LIN {X 0,Y 523.443,Z 553.477,A -85,B 0,C 180,E1 -4766.15,E2 -4766.15} C_VEL
LIN {X 0,Y 523.367,Z 555.34,A -85,B 0,C 180,E1 -4766.921,E2 -4766.921} C_VEL
LIN {X 0,Y 523.334,Z 556.738,A -85,B 0,C 180,E1 -4767.691,E2 -4767.691} C_VEL
LIN {X 0,Y 523.25,Z 558.344,A -85,B 0,C 180,E1 -4769.23,E2 -4769.23} C_VEL
LIN {X 0,Y 523.25,Z 558.561,A -85,B 0,C 180,E1 -4770,E2 -4770} C_VEL
LIN {X 0,Y 523.274,Z 557.739,A -85,B 0,C 180,E1 -4771.539,E2 -4771.539} C_VEL
LIN {X 0,Y 523.334,Z 556.745,A -85,B 0,C 180,E1 -4772.309,E2 -4772.309} C_VEL
LIN {X 0,Y 523.367,Z 555.349,A -85,B 0,C 180,E1 -4773.079,E2 -4773.079} C_VEL
LIN {X 0,Y 523.424,Z 552.411,A -85,B 0,C 180,E1 -4774.235,E2 -4774.235} C_VEL
LIN {X 0,Y 523.461,Z 548.432,A -85,B 0,C 180,E1 -4775.392,E2 -4775.392} C_VEL
LIN {X 0,Y 523.514,Z 543.213,A -85,B 0,C 180,E1 -4776.572,E2 -4776.572} C_VEL
LIN {X 0,Y 523.646,Z 536.865,A -85,B 0,C 180,E1 -4777.713,E2 -4777.713} C_VEL
LIN {X 0,Y 523.815,Z 528.823,A -85,B 0,C 180,E1 -4778.876,E2 -4778.876} C_VEL
LIN {X 0,Y 524.043,Z 520.63,A -85,B 0,C 180,E1 -4779.845,E2 -4779.845} C_VEL
LIN {X 0,Y 524.325,Z 510.642,A -85,B 0,C 180,E1 -4780.816,E2 -4780.816} C_VEL
LIN {X 0,Y 524.62,Z 499.343,A -85,B 0,C 180,E1 -4781.691,E2 -4781.691} C_VEL
LIN {X 0,Y 524.85,Z 488.315,A -85,B 0,C 180,E1 -4782.371,E2 -4782.371} C_VEL
LIN {X 0,Y 525.116,Z 476.074,A -85,B 0,C 180,E1 -4782.954,E2 -4782.954} C_VEL
LIN {X 0,Y 525.355,Z 463.228,A -85,B 0,C 180,E1 -4783.391,E2 -4783.391} C_VEL
LIN {X 0,Y 525.545,Z 449.606,A -85,B 0,C 180,E1 -4783.681,E2 -4783.681} C_VEL
LIN {X 0,Y 525.885,Z 356.541,A -85,B 0,C 180,E1 -4784.961,E2 -4784.961} C_VEL
LIN {X 0,Y 524.307,Z 345.556,A -85,B 0,C 180,E1 -4785.178,E2 -4785.178} C_VEL
LIN {X 0,Y 524.738,Z 323.578,A -85,B 0,C 180,E1 -4788.527,E2 -4788.527} C_VEL
LIN {X 0,Y 525.158,Z 305.074,A -85,B 0,C 180,E1 -4791.387,E2 -4791.387} C_VEL
LIN {X 0,Y 525.431,Z 293.248,A -85,B 0,C 180,E1 -4793.239,E2 -4793.239} C_VEL
LIN {X 0,Y 524.002,Z 285.214,A -85,B 0,C 180,E1 -4794.594,E2 -4794.594} C_VEL
LIN {X 0,Y 523.979,Z 285.218,A -85,B 0,C 180,E1 -4797.718,E2 -4797.718} C_VEL
LIN {X 0,Y 523.945,Z 285.215,A -85,B 0,C 180,E1 -4800.854,E2 -4800.854} C_VEL
LIN {X 0,Y 523.959,Z 285.215,A -85,B 0,C 180,E1 -4803.734,E2 -4803.734} C_VEL
LIN {X 0,Y 523.903,Z 285.227,A -85,B 0,C 180,E1 -4806.401,E2 -4806.401} C_VEL
LIN {X 0,Y 523.919,Z 285.218,A -85,B 0,C 180,E1 -4809.084,E2 -4809.084} C_VEL
LIN {X 0,Y 523.953,Z 285.218,A -85,B 0,C 180,E1 -4812.118,E2 -4812.118} C_VEL
LIN {X 0,Y 523.942,Z 285.215,A -85,B 0,C 180,E1 -4815.309,E2 -4815.309} C_VEL
LIN {X 0,Y 523.957,Z 285.221,A -85,B 0,C 180,E1 -4818.689,E2 -4818.689} C_VEL
LIN {X 0,Y 523.914,Z 285.221,A -85,B 0,C 180,E1 -4821.08,E2 -4821.08} C_VEL
LIN {X 0,Y 523.898,Z 285.22,A -85,B 0,C 180,E1 -4823.825,E2 -4823.825} C_VEL
LIN {X 0,Y 523.938,Z 285.222,A -85,B 0,C 180,E1 -4826.635,E2 -4826.635} C_VEL
LIN {X 0,Y 523.953,Z 285.216,A -85,B 0,C 180,E1 -4829.355,E2 -4829.355} C_VEL
LIN {X 0,Y 523.975,Z 285.211,A -85,B 0,C 180,E1 -4832.281,E2 -4832.281} C_VEL
LIN {X 0,Y 523.949,Z 285.217,A -85,B 0,C 180,E1 -4834.581,E2 -4834.581} C_VEL
LIN {X 0,Y 523.913,Z 285.228,A -85,B 0,C 180,E1 -4837.106,E2 -4837.106} C_VEL
LIN {X 0,Y 523.974,Z 285.211,A -85,B 0,C 180,E1 -4839.866,E2 -4839.866} C_VEL
LIN {X 0,Y 523.962,Z 285.215,A -85,B 0,C 180,E1 -4842.837,E2 -4842.837} C_VEL
LIN {X 0,Y 524,Z 285.216,A -85,B 0,C 180,E1 -4845.236,E2 -4845.236} C_VEL
LIN {X 0,Y 524.007,Z 285.206,A -85,B 0,C 180,E1 -4848.394,E2 -4848.394} C_VEL
LIN {X 0,Y 524,Z 285.217,A -85,B 0,C 180,E1 -4851.516,E2 -4851.516} C_VEL
LIN {X 0,Y 524.076,Z 285.198,A -85,B 0,C 180,E1 -4854.613,E2 -4854.613} C_VEL
LIN {X 0,Y 524.104,Z 285.204,A -85,B 0,C 180,E1 -4857.694,E2 -4857.694} C_VEL
LIN {X 0,Y 524.116,Z 285.193,A -85,B 0,C 180,E1 -4860.768,E2 -4860.768} C_VEL
LIN {X 0,Y 524.067,Z 285.2,A -85,B 0,C 180,E1 -4863.075,E2 -4863.075} C_VEL
LIN {X 0,Y 524.023,Z 285.21,A -85,B 0,C 180,E1 -4866.159,E2 -4866.159} C_VEL
LIN {X 0,Y 523.998,Z 285.21,A -85,B 0,C 180,E1 -4868.484,E2 -4868.484} C_VEL
LIN {X 0,Y 523.997,Z 285.213,A -85,B 0,C 180,E1 -4871.739,E2 -4871.739} C_VEL
LIN {X 0,Y 523.986,Z 285.209,A -85,B 0,C 180,E1 -4875.052,E2 -4875.052} C_VEL
LIN {X 0,Y 523.941,Z 285.22,A -85,B 0,C 180,E1 -4877.97,E2 -4877.97} C_VEL
LIN {X 0,Y 523.966,Z 285.219,A -85,B 0,C 180,E1 -4880.41,E2 -4880.41} C_VEL
LIN {X 0,Y 523.904,Z 285.221,A -85,B 0,C 180,E1 -4882.894,E2 -4882.894} C_VEL
LIN {X 0,Y 523.977,Z 285.214,A -85,B 0,C 180,E1 -4886.02,E2 -4886.02} C_VEL
LIN {X 0,Y 523.927,Z 285.22,A -85,B 0,C 180,E1 -4888.875,E2 -4888.875} C_VEL
LIN {X 0,Y 523.915,Z 285.218,A -85,B 0,C 180,E1 -4891.544,E2 -4891.544} C_VEL
LIN {X 0,Y 523.927,Z 285.22,A -85,B 0,C 180,E1 -4894.291,E2 -4894.291} C_VEL
LIN {X 0,Y 523.901,Z 285.223,A -85,B 0,C 180,E1 -4897.133,E2 -4897.133} C_VEL
LIN {X 0,Y 523.933,Z 285.216,A -85,B 0,C 180,E1 -4900.13,E2 -4900.13} C_VEL
LIN {X 0,Y 523.93,Z 285.219,A -85,B 0,C 180,E1 -4902.459,E2 -4902.459} C_VEL
LIN {X 0,Y 523.948,Z 285.218,A -85,B 0,C 180,E1 -4905.31,E2 -4905.31} C_VEL
LIN {X 0,Y 523.891,Z 285.227,A -85,B 0,C 180,E1 -4906.893,E2 -4906.893} C_VEL
LIN {X 0,Y 523.211,Z 285.309,A -85,B 0,C 180,E1 -4907.535,E2 -4907.535} C_VEL
LIN {X 0,Y 520.359,Z 285.664,A -85,B 0,C 180,E1 -4908.576,E2 -4908.576} C_VEL
LIN {X 0,Y 517.961,Z 285.964,A -85,B 0,C 180,E1 -4909.415,E2 -4909.415} C_VEL
LIN {X 0,Y 516.935,Z 286.088,A -85,B 0,C 180,E1 -4910.063,E2 -4910.063} C_VEL
LIN {X 0,Y 516.854,Z 286.098,A -85,B 0,C 180,E1 -4910.282,E2 -4910.282} C_VEL
LIN {X 0,Y 516.873,Z 286.102,A -85,B 0,C 180,E1 -4913.344,E2 -4913.344} C_VEL
LIN {X 0,Y 516.88,Z 286.094,A -85,B 0,C 180,E1 -4916.119,E2 -4916.119} C_VEL
LIN {X 0,Y 516.885,Z 286.097,A -85,B 0,C 180,E1 -4918.937,E2 -4918.937} C_VEL
LIN {X 0,Y 516.855,Z 286.104,A -85,B 0,C 180,E1 -4921.582,E2 -4921.582} C_VEL
LIN {X 0,Y 516.865,Z 286.097,A -85,B 0,C 180,E1 -4924.208,E2 -4924.208} C_VEL
LIN {X 0,Y 516.855,Z 286.098,A -85,B 0,C 180,E1 -4926.776,E2 -4926.776} C_VEL
LIN {X 0,Y 516.938,Z 286.095,A -85,B 0,C 180,E1 -4929.732,E2 -4929.732} C_VEL
LIN {X 0,Y 516.883,Z 286.094,A -85,B 0,C 180,E1 -4932.595,E2 -4932.595} C_VEL
LIN {X 0,Y 516.941,Z 286.087,A -85,B 0,C 180,E1 -4935.031,E2 -4935.031} C_VEL
LIN {X 0,Y 516.925,Z 286.096,A -85,B 0,C 180,E1 -4938.233,E2 -4938.233} C_VEL
LIN {X 0,Y 516.906,Z 286.192,A -85,B 0,C 180,E1 -4940.289,E2 -4940.289} C_VEL
LIN {X 0,Y 517.467,Z 290.917,A -85,B 0,C 180,E1 -4941.212,E2 -4941.212} C_VEL
LIN {X 0,Y 517.225,Z 306.513,A -85,B 0,C 180,E1 -4944.151,E2 -4944.151} C_VEL
LIN {X 0,Y 517.209,Z 309.369,A -85,B 0,C 180,E1 -4944.689,E2 -4944.689} C_VEL
LIN {X 0,Y 519.108,Z 320.246,A -85,B 0,C 180,E1 -4944.903,E2 -4944.903} C_VEL
LIN {X 0,Y 518.613,Z 416.523,A -85,B 0,C 180,E1 -4946.261,E2 -4946.261} C_VEL
LIN {X 0,Y 518.43,Z 429.494,A -85,B 0,C 180,E1 -4946.6,E2 -4946.6} C_VEL
LIN {X 0,Y 518.257,Z 441.97,A -85,B 0,C 180,E1 -4947.085,E2 -4947.085} C_VEL
LIN {X 0,Y 517.976,Z 453.153,A -85,B 0,C 180,E1 -4947.667,E2 -4947.667} C_VEL
LIN {X 0,Y 517.599,Z 464.695,A -85,B 0,C 180,E1 -4948.444,E2 -4948.444} C_VEL
LIN {X 0,Y 517.235,Z 475.076,A -85,B 0,C 180,E1 -4949.319,E2 -4949.319} C_VEL
LIN {X 0,Y 517.081,Z 483.55,A -85,B 0,C 180,E1 -4950.195,E2 -4950.195} C_VEL
LIN {X 0,Y 516.841,Z 491.401,A -85,B 0,C 180,E1 -4951.169,E2 -4951.169} C_VEL
LIN {X 0,Y 516.597,Z 499.125,A -85,B 0,C 180,E1 -4952.339,E2 -4952.339} C_VEL
LIN {X 0,Y 516.472,Z 505.306,A -85,B 0,C 180,E1 -4953.511,E2 -4953.511} C_VEL
LIN {X 0,Y 516.328,Z 510.245,A -85,B 0,C 180,E1 -4954.685,E2 -4954.685} C_VEL
LIN {X 0,Y 516.374,Z 514.064,A -85,B 0,C 180,E1 -4955.859,E2 -4955.859} C_VEL
LIN {X 0,Y 516.281,Z 516.886,A -85,B 0,C 180,E1 -4957.037,E2 -4957.037} C_VEL
LIN {X 0,Y 516.266,Z 518.217,A -85,B 0,C 180,E1 -4957.824,E2 -4957.824} C_VEL
LIN {X 0,Y 516.212,Z 519.159,A -85,B 0,C 180,E1 -4958.613,E2 -4958.613} C_VEL
LIN {X 0,Y 516.175,Z 519.709,A -85,B 0,C 180,E1 -4959.404,E2 -4959.404} C_VEL
LIN {X 0,Y 516.236,Z 519.817,A -85,B 0,C 180,E1 -4960.194,E2 -4960.194} C_VEL
LIN {X 0,Y 516.281,Z 519.192,A -85,B 0,C 180,E1 -4961.445,E2 -4961.445} C_VEL
LIN {X 0,Y 516.223,Z 517.759,A -85,B 0,C 180,E1 -4962.582,E2 -4962.582} C_VEL
LIN {X 0,Y 516.234,Z 516.198,A -85,B 0,C 180,E1 -4963.382,E2 -4963.382} C_VEL
LIN {X 0,Y 516.359,Z 513.134,A -85,B 0,C 180,E1 -4964.553,E2 -4964.553} C_VEL
LIN {X 0,Y 516.416,Z 508.746,A -85,B 0,C 180,E1 -4965.794,E2 -4965.794} C_VEL
LIN {X 0,Y 516.554,Z 503.194,A -85,B 0,C 180,E1 -4967.009,E2 -4967.009} C_VEL
LIN {X 0,Y 516.753,Z 496.184,A -85,B 0,C 180,E1 -4968.229,E2 -4968.229} C_VEL
LIN {X 0,Y 516.9,Z 488.946,A -85,B 0,C 180,E1 -4969.252,E2 -4969.252} C_VEL
LIN {X 0,Y 517.195,Z 479.415,A -85,B 0,C 180,E1 -4970.345,E2 -4970.345} C_VEL
LIN {X 0,Y 517.499,Z 469.068,A -85,B 0,C 180,E1 -4971.302,E2 -4971.302} C_VEL
LIN {X 0,Y 517.853,Z 457.976,A -85,B 0,C 180,E1 -4972.124,E2 -4972.124} C_VEL
LIN {X 0,Y 518.12,Z 446.531,A -85,B 0,C 180,E1 -4972.787,E2 -4972.787} C_VEL
LIN {X 0,Y 518.289,Z 434.594,A -85,B 0,C 180,E1 -4973.315,E2 -4973.315} C_VEL
LIN {X 0,Y 518.439,Z 421.216,A -85,B 0,C 180,E1 -4973.731,E2 -4973.731} C_VEL
LIN {X 0,Y 518.604,Z 406.66,A -85,B 0,C 180,E1 -4973.989,E2 -4973.989} C_VEL
LIN {X 0,Y 519.054,Z 319.507,A -85,B 0,C 180,E1 -4975.2,E2 -4975.2} C_VEL
LIN {X 0,Y 517.236,Z 309.202,A -85,B 0,C 180,E1 -4975.422,E2 -4975.422} C_VEL
LIN {X 0,Y 517.357,Z 293.041,A -85,B 0,C 180,E1 -4978.389,E2 -4978.389} C_VEL
LIN {X 0,Y 517.28,Z 288.195,A -85,B 0,C 180,E1 -4979.282,E2 -4979.282} C_VEL
LIN {X 0,Y 516.952,Z 286.097,A -85,B 0,C 180,E1 -4979.697,E2 -4979.697} C_VEL
LIN {X 0,Y 516.894,Z 286.096,A -85,B 0,C 180,E1 -4982.947,E2 -4982.947} C_VEL
LIN {X 0,Y 516.871,Z 286.099,A -85,B 0,C 180,E1 -4985.78,E2 -4985.78} C_VEL
LIN {X 0,Y 516.879,Z 286.102,A -85,B 0,C 180,E1 -4988.716,E2 -4988.716} C_VEL
LIN {X 0,Y 516.911,Z 286.092,A -85,B 0,C 180,E1 -4991.775,E2 -4991.775} C_VEL
LIN {X 0,Y 516.894,Z 286.098,A -85,B 0,C 180,E1 -4995.007,E2 -4995.007} C_VEL
LIN {X 0,Y 516.912,Z 286.095,A -85,B 0,C 180,E1 -4998.399,E2 -4998.399} C_VEL
LIN {X 0,Y 516.88,Z 286.097,A -85,B 0,C 180,E1 -5001.284,E2 -5001.284} C_VEL
LIN {X 0,Y 516.87,Z 286.095,A -85,B 0,C 180,E1 -5004.22,E2 -5004.22} C_VEL
LIN {X 0,Y 516.894,Z 286.1,A -85,B 0,C 180,E1 -5007.053,E2 -5007.053} C_VEL
LIN {X 0,Y 516.891,Z 286.092,A -85,B 0,C 180,E1 -5009.796,E2 -5009.796} C_VEL
LIN {X 0,Y 516.925,Z 286.087,A -85,B 0,C 180,E1 -5012.467,E2 -5012.467} C_VEL
LIN {X 0,Y 516.908,Z 286.096,A -85,B 0,C 180,E1 -5015.072,E2 -5015.072} C_VEL
LIN {X 0,Y 516.884,Z 286.093,A -85,B 0,C 180,E1 -5018.462,E2 -5018.462} C_VEL
LIN {X 0,Y 516.9,Z 286.092,A -85,B 0,C 180,E1 -5020.955,E2 -5020.955} C_VEL
LIN {X 0,Y 516.913,Z 286.099,A -85,B 0,C 180,E1 -5023.41,E2 -5023.41} C_VEL
LIN {X 0,Y 516.894,Z 286.099,A -85,B 0,C 180,E1 -5025.834,E2 -5025.834} C_VEL
LIN {X 0,Y 516.965,Z 286.084,A -85,B 0,C 180,E1 -5028.234,E2 -5028.234} C_VEL
LIN {X 0,Y 516.967,Z 286.088,A -85,B 0,C 180,E1 -5031.4,E2 -5031.4} C_VEL
LIN {X 0,Y 517.001,Z 286.086,A -85,B 0,C 180,E1 -5033.757,E2 -5033.757} C_VEL
LIN {X 0,Y 517.012,Z 286.077,A -85,B 0,C 180,E1 -5036.883,E2 -5036.883} C_VEL
LIN {X 0,Y 517.085,Z 286.077,A -85,B 0,C 180,E1 -5040,E2 -5040} C_VEL
LIN {X 0,Y 517.012,Z 286.076,A -85,B 0,C 180,E1 -5043.117,E2 -5043.117} C_VEL
LIN {X 0,Y 517.002,Z 286.085,A -85,B 0,C 180,E1 -5046.243,E2 -5046.243} C_VEL
LIN {X 0,Y 516.951,Z 286.085,A -85,B 0,C 180,E1 -5049.389,E2 -5049.389} C_VEL
LIN {X 0,Y 516.951,Z 286.084,A -85,B 0,C 180,E1 -5051.807,E2 -5051.807} C_VEL
LIN {X 0,Y 516.944,Z 286.086,A -85,B 0,C 180,E1 -5055.147,E2 -5055.147} C_VEL
LIN {X 0,Y 516.924,Z 286.092,A -85,B 0,C 180,E1 -5058.222,E2 -5058.222} C_VEL
LIN {X 0,Y 516.912,Z 286.097,A -85,B 0,C 180,E1 -5060.702,E2 -5060.702} C_VEL
LIN {X 0,Y 516.904,Z 286.092,A -85,B 0,C 180,E1 -5064.073,E2 -5064.073} C_VEL
LIN {X 0,Y 516.925,Z 286.095,A -85,B 0,C 180,E1 -5066.658,E2 -5066.658} C_VEL
LIN {X 0,Y 516.911,Z 286.092,A -85,B 0,C 180,E1 -5069.524,E2 -5069.524} C_VEL
LIN {X 0,Y 516.896,Z 286.094,A -85,B 0,C 180,E1 -5072.544,E2 -5072.544} C_VEL
LIN {X 0,Y 516.866,Z 286.101,A -85,B 0,C 180,E1 -5075.33,E2 -5075.33} C_VEL
LIN {X 0,Y 516.881,Z 286.095,A -85,B 0,C 180,E1 -5077.943,E2 -5077.943} C_VEL
LIN {X 0,Y 516.884,Z 286.09,A -85,B 0,C 180,E1 -5080.742,E2 -5080.742} C_VEL
LIN {X 0,Y 516.883,Z 286.096,A -85,B 0,C 180,E1 -5082.832,E2 -5082.832} C_VEL
LIN {X 0,Y 516.896,Z 286.095,A -85,B 0,C 180,E1 -5085.007,E2 -5085.007} C_VEL
LIN {X 0,Y 516.915,Z 286.091,A -85,B 0,C 180,E1 -5088.399,E2 -5088.399} C_VEL
LIN {X 0,Y 516.882,Z 286.099,A -85,B 0,C 180,E1 -5091.284,E2 -5091.284} C_VEL
LIN {X 0,Y 516.873,Z 286.099,A -85,B 0,C 180,E1 -5094.22,E2 -5094.22} C_VEL
LIN {X 0,Y 516.897,Z 286.095,A -85,B 0,C 180,E1 -5097.053,E2 -5097.053} C_VEL
LIN {X 0,Y 516.895,Z 286.101,A -85,B 0,C 180,E1 -5099.796,E2 -5099.796} C_VEL
LIN {X 0,Y 516.926,Z 286.093,A -85,B 0,C 180,E1 -5102.467,E2 -5102.467} C_VEL
LIN {X 0,Y 516.938,Z 286.123,A -85,B 0,C 180,E1 -5105.295,E2 -5105.295} C_VEL
LIN {X 0,Y 518.392,Z 294.033,A -85,B 0,C 180,E1 -5106.637,E2 -5106.637} C_VEL
LIN {X 0,Y 518.071,Z 309.859,A -85,B 0,C 180,E1 -5109.139,E2 -5109.139} C_VEL
LIN {X 0,Y 517.59,Z 329.884,A -85,B 0,C 180,E1 -5112.251,E2 -5112.251} C_VEL
LIN {X 0,Y 517.286,Z 345.547,A -85,B 0,C 180,E1 -5114.634,E2 -5114.634} C_VEL
LIN {X 0,Y 519.046,Z 357.722,A -85,B 0,C 180,E1 -5114.858,E2 -5114.858} C_VEL
LIN {X 0,Y 518.595,Z 453.618,A -85,B 0,C 180,E1 -5116.206,E2 -5116.206} C_VEL
LIN {X 0,Y 518.365,Z 466.951,A -85,B 0,C 180,E1 -5116.549,E2 -5116.549} C_VEL
LIN {X 0,Y 518.053,Z 480.278,A -85,B 0,C 180,E1 -5117.065,E2 -5117.065} C_VEL
LIN {X 0,Y 517.807,Z 492.339,A -85,B 0,C 180,E1 -5117.711,E2 -5117.711} C_VEL
LIN {X 0,Y 517.514,Z 504.391,A -85,B 0,C 180,E1 -5118.544,E2 -5118.544} C_VEL
LIN {X 0,Y 517.17,Z 514.61,A -85,B 0,C 180,E1 -5119.429,E2 -5119.429} C_VEL
LIN {X 0,Y 516.891,Z 523.806,A -85,B 0,C 180,E1 -5120.412,E2 -5120.412} C_VEL
LIN {X 0,Y 516.658,Z 532.769,A -85,B 0,C 180,E1 -5121.591,E2 -5121.591} C_VEL
LIN {X 0,Y 516.505,Z 539.985,A -85,B 0,C 180,E1 -5122.769,E2 -5122.769} C_VEL
LIN {X 0,Y 516.419,Z 546.558,A -85,B 0,C 180,E1 -5124.141,E2 -5124.141} C_VEL
LIN {X 0,Y 516.269,Z 550.903,A -85,B 0,C 180,E1 -5125.315,E2 -5125.315} C_VEL
LIN {X 0,Y 516.352,Z 553.21,A -85,B 0,C 180,E1 -5126.098,E2 -5126.098} C_VEL
LIN {X 0,Y 516.282,Z 555.074,A -85,B 0,C 180,E1 -5126.878,E2 -5126.878} C_VEL
LIN {X 0,Y 516.261,Z 556.473,A -85,B 0,C 180,E1 -5127.659,E2 -5127.659} C_VEL
LIN {X 0,Y 516.16,Z 558.079,A -85,B 0,C 180,E1 -5129.22,E2 -5129.22} C_VEL
LIN {X 0,Y 516.158,Z 558.297,A -85,B 0,C 180,E1 -5130,E2 -5130} C_VEL
LIN {X 0,Y 516.191,Z 557.476,A -85,B 0,C 180,E1 -5131.56,E2 -5131.56} C_VEL
LIN {X 0,Y 516.26,Z 556.482,A -85,B 0,C 180,E1 -5132.34,E2 -5132.34} C_VEL
LIN {X 0,Y 516.282,Z 555.086,A -85,B 0,C 180,E1 -5133.121,E2 -5133.121} C_VEL
LIN {X 0,Y 516.312,Z 552.147,A -85,B 0,C 180,E1 -5134.293,E2 -5134.293} C_VEL
LIN {X 0,Y 516.375,Z 548.168,A -85,B 0,C 180,E1 -5135.467,E2 -5135.467} C_VEL
LIN {X 0,Y 516.45,Z 542.253,A -85,B 0,C 180,E1 -5136.798,E2 -5136.798} C_VEL
LIN {X 0,Y 516.597,Z 535.359,A -85,B 0,C 180,E1 -5138.015,E2 -5138.015} C_VEL
LIN {X 0,Y 516.811,Z 527.063,A -85,B 0,C 180,E1 -5139.194,E2 -5139.194} C_VEL
LIN {X 0,Y 517.039,Z 518.559,A -85,B 0,C 180,E1 -5140.178,E2 -5140.178} C_VEL
LIN {X 0,Y 517.367,Z 508.054,A -85,B 0,C 180,E1 -5141.161,E2 -5141.161} C_VEL
LIN {X 0,Y 517.712,Z 496.59,A -85,B 0,C 180,E1 -5142.022,E2 -5142.022} C_VEL
LIN {X 0,Y 517.952,Z 486.272,A -85,B 0,C 180,E1 -5142.638,E2 -5142.638} C_VEL
LIN {X 0,Y 518.211,Z 474.582,A -85,B 0,C 180,E1 -5143.18,E2 -5143.18} C_VEL
LIN {X 0,Y 518.47,Z 461.116,A -85,B 0,C 180,E1 -5143.622,E2 -5143.622} C_VEL
LIN {X 0,Y 518.663,Z 447.786,A -85,B 0,C 180,E1 -5143.892,E2 -5143.892} C_VEL
LIN {X 0,Y 519.011,Z 357.28,A -85,B 0,C 180,E1 -5145.15,E2 -5145.15} C_VEL
LIN {X 0,Y 517.275,Z 345.369,A -85,B 0,C 180,E1 -5145.377,E2 -5145.377} C_VEL
LIN {X 0,Y 517.743,Z 324.502,A -85,B 0,C 180,E1 -5148.602,E2 -5148.602} C_VEL
LIN {X 0,Y 518.196,Z 306.136,A -85,B 0,C 180,E1 -5151.48,E2 -5151.48} C_VEL
LIN {X 0,Y 518.447,Z 294.291,A -85,B 0,C 180,E1 -5153.36,E2 -5153.36} C_VEL
LIN {X 0,Y 516.94,Z 286.093,A -85,B 0,C 180,E1 -5154.781,E2 -5154.781} C_VEL
LIN {X 0,Y 516.927,Z 286.098,A -85,B 0,C 180,E1 -5157.905,E2 -5157.905} C_VEL
LIN {X 0,Y 516.892,Z 286.103,A -85,B 0,C 180,E1 -5160.203,E2 -5160.203} C_VEL
LIN {X 0,Y 516.894,Z 286.093,A -85,B 0,C 180,E1 -5162.946,E2 -5162.946} C_VEL
LIN {X 0,Y 516.87,Z 286.098,A -85,B 0,C 180,E1 -5165.78,E2 -5165.78} C_VEL
LIN {X 0,Y 516.879,Z 286.098,A -85,B 0,C 180,E1 -5168.715,E2 -5168.715} C_VEL
LIN {X 0,Y 516.912,Z 286.091,A -85,B 0,C 180,E1 -5171.774,E2 -5171.774} C_VEL
LIN {X 0,Y 516.893,Z 286.095,A -85,B 0,C 180,E1 -5175.006,E2 -5175.006} C_VEL
LIN {X 0,Y 516.913,Z 286.097,A -85,B 0,C 180,E1 -5178.398,E2 -5178.398} C_VEL
LIN {X 0,Y 516.877,Z 286.096,A -85,B 0,C 180,E1 -5181.284,E2 -5181.284} C_VEL
LIN {X 0,Y 516.869,Z 286.098,A -85,B 0,C 180,E1 -5184.219,E2 -5184.219} C_VEL
LIN {X 0,Y 516.891,Z 286.099,A -85,B 0,C 180,E1 -5187.053,E2 -5187.053} C_VEL
LIN {X 0,Y 516.889,Z 286.093,A -85,B 0,C 180,E1 -5189.796,E2 -5189.796} C_VEL
LIN {X 0,Y 516.924,Z 286.091,A -85,B 0,C 180,E1 -5192.467,E2 -5192.467} C_VEL
LIN {X 0,Y 516.907,Z 286.101,A -85,B 0,C 180,E1 -5195.071,E2 -5195.071} C_VEL
LIN {X 0,Y 516.865,Z 286.098,A -85,B 0,C 180,E1 -5197.621,E2 -5197.621} C_VEL
LIN {X 0,Y 516.927,Z 286.088,A -85,B 0,C 180,E1 -5200.129,E2 -5200.129} C_VEL
LIN {X 0,Y 516.924,Z 286.09,A -85,B 0,C 180,E1 -5202.596,E2 -5202.596} C_VEL
LIN {X 0,Y 516.946,Z 286.091,A -85,B 0,C 180,E1 -5205.03,E2 -5205.03} C_VEL
LIN {X 0,Y 516.961,Z 286.084,A -85,B 0,C 180,E1 -5208.233,E2 -5208.233} C_VEL
LIN {X 0,Y 516.965,Z 286.092,A -85,B 0,C 180,E1 -5211.399,E2 -5211.399} C_VEL
LIN {X 0,Y 516.997,Z 286.086,A -85,B 0,C 180,E1 -5213.756,E2 -5213.756} C_VEL
LIN {X 0,Y 517.008,Z 286.079,A -85,B 0,C 180,E1 -5216.883,E2 -5216.883} C_VEL
LIN {X 0,Y 517.078,Z 286.075,A -85,B 0,C 180,E1 -5220,E2 -5220} C_VEL
LIN {X 0,Y 517.008,Z 286.079,A -85,B 0,C 180,E1 -5223.117,E2 -5223.117} C_VEL
LIN {X 0,Y 516.985,Z 286.085,A -85,B 0,C 180,E1 -5226.243,E2 -5226.243} C_VEL
LIN {X 0,Y 516.963,Z 286.085,A -85,B 0,C 180,E1 -5228.6,E2 -5228.6} C_VEL
LIN {X 0,Y 516.946,Z 286.092,A -85,B 0,C 180,E1 -5231.807,E2 -5231.807} C_VEL
LIN {X 0,Y 516.937,Z 286.087,A -85,B 0,C 180,E1 -5235.146,E2 -5235.146} C_VEL
LIN {X 0,Y 516.91,Z 286.101,A -85,B 0,C 180,E1 -5238.223,E2 -5238.223} C_VEL
LIN {X 0,Y 516.906,Z 286.094,A -85,B 0,C 180,E1 -5240.702,E2 -5240.702} C_VEL
LIN {X 0,Y 516.885,Z 286.098,A -85,B 0,C 180,E1 -5244.073,E2 -5244.073} C_VEL
LIN {X 0,Y 516.912,Z 286.097,A -85,B 0,C 180,E1 -5246.658,E2 -5246.658} C_VEL
LIN {X 0,Y 516.905,Z 286.091,A -85,B 0,C 180,E1 -5249.524,E2 -5249.524} C_VEL
LIN {X 0,Y 516.89,Z 286.102,A -85,B 0,C 180,E1 -5252.544,E2 -5252.544} C_VEL
LIN {X 0,Y 516.86,Z 286.098,A -85,B 0,C 180,E1 -5255.33,E2 -5255.33} C_VEL
LIN {X 0,Y 516.874,Z 286.095,A -85,B 0,C 180,E1 -5257.943,E2 -5257.943} C_VEL
LIN {X 0,Y 516.878,Z 286.103,A -85,B 0,C 180,E1 -5260.742,E2 -5260.742} C_VEL
LIN {X 0,Y 516.878,Z 286.104,A -85,B 0,C 180,E1 -5262.832,E2 -5262.832} C_VEL
LIN {X 0,Y 516.919,Z 286.098,A -85,B 0,C 180,E1 -5265.01,E2 -5265.01} C_VEL
LIN {X 0,Y 516.883,Z 286.095,A -85,B 0,C 180,E1 -5268.402,E2 -5268.402} C_VEL
LIN {X 0,Y 516.854,Z 286.098,A -85,B 0,C 180,E1 -5270.282,E2 -5270.282} C_VEL
LIN {X 0,Y 516.196,Z 286.187,A -85,B 0,C 180,E1 -5270.932,E2 -5270.932} C_VEL
LIN {X 0,Y 513.36,Z 286.54,A -85,B 0,C 180,E1 -5271.988,E2 -5271.988} C_VEL
LIN {X 0,Y 510.952,Z 286.84,A -85,B 0,C 180,E1 -5272.839,E2 -5272.839} C_VEL
LIN {X 0,Y 509.907,Z 286.968,A -85,B 0,C 180,E1 -5273.495,E2 -5273.495} C_VEL
LIN {X 0,Y 509.817,Z 286.976,A -85,B 0,C 180,E1 -5273.718,E2 -5273.718} C_VEL
LIN {X 0,Y 509.838,Z 286.972,A -85,B 0,C 180,E1 -5276.538,E2 -5276.538} C_VEL
LIN {X 0,Y 509.831,Z 286.982,A -85,B 0,C 180,E1 -5279.334,E2 -5279.334} C_VEL
LIN {X 0,Y 509.834,Z 286.973,A -85,B 0,C 180,E1 -5282.052,E2 -5282.052} C_VEL
LIN {X 0,Y 509.797,Z 286.977,A -85,B 0,C 180,E1 -5284.7,E2 -5284.7} C_VEL
LIN {X 0,Y 509.824,Z 286.981,A -85,B 0,C 180,E1 -5287.459,E2 -5287.459} C_VEL
LIN {X 0,Y 509.915,Z 286.968,A -85,B 0,C 180,E1 -5289.845,E2 -5289.845} C_VEL
LIN {X 0,Y 509.854,Z 286.971,A -85,B 0,C 180,E1 -5293.174,E2 -5293.174} C_VEL
LIN {X 0,Y 509.857,Z 286.976,A -85,B 0,C 180,E1 -5295.634,E2 -5295.634} C_VEL
LIN {X 0,Y 509.888,Z 286.974,A -85,B 0,C 180,E1 -5298.131,E2 -5298.131} C_VEL
LIN {X 0,Y 509.885,Z 287.126,A -85,B 0,C 180,E1 -5300.179,E2 -5300.179} C_VEL
LIN {X 0,Y 510.476,Z 291.744,A -85,B 0,C 180,E1 -5301.09,E2 -5301.09} C_VEL
LIN {X 0,Y 510.224,Z 307.449,A -85,B 0,C 180,E1 -5304.071,E2 -5304.071} C_VEL
LIN {X 0,Y 510.178,Z 309.558,A -85,B 0,C 180,E1 -5304.467,E2 -5304.467} C_VEL
LIN {X 0,Y 512.283,Z 321.57,A -85,B 0,C 180,E1 -5304.712,E2 -5304.712} C_VEL
LIN {X 0,Y 511.76,Z 416.317,A -85,B 0,C 180,E1 -5306.063,E2 -5306.063} C_VEL
LIN {X 0,Y 511.541,Z 429.46,A -85,B 0,C 180,E1 -5306.406,E2 -5306.406} C_VEL
LIN {X 0,Y 511.359,Z 442.009,A -85,B 0,C 180,E1 -5306.898,E2 -5306.898} C_VEL
LIN {X 0,Y 511.027,Z 454.052,A -85,B 0,C 180,E1 -5307.537,E2 -5307.537} C_VEL
LIN {X 0,Y 510.62,Z 465.471,A -85,B 0,C 180,E1 -5308.324,E2 -5308.324} C_VEL
LIN {X 0,Y 510.246,Z 475.762,A -85,B 0,C 180,E1 -5309.211,E2 -5309.211} C_VEL
LIN {X 0,Y 510.047,Z 485.032,A -85,B 0,C 180,E1 -5310.198,E2 -5310.198} C_VEL
LIN {X 0,Y 509.755,Z 494.007,A -85,B 0,C 180,E1 -5311.383,E2 -5311.383} C_VEL
LIN {X 0,Y 509.528,Z 501.263,A -85,B 0,C 180,E1 -5312.57,E2 -5312.57} C_VEL
LIN {X 0,Y 509.356,Z 507.944,A -85,B 0,C 180,E1 -5313.956,E2 -5313.956} C_VEL
LIN {X 0,Y 509.246,Z 512.368,A -85,B 0,C 180,E1 -5315.147,E2 -5315.147} C_VEL
LIN {X 0,Y 509.286,Z 516.079,A -85,B 0,C 180,E1 -5316.497,E2 -5316.497} C_VEL
LIN {X 0,Y 509.169,Z 518.679,A -85,B 0,C 180,E1 -5317.934,E2 -5317.934} C_VEL
LIN {X 0,Y 509.119,Z 519.564,A -85,B 0,C 180,E1 -5318.734,E2 -5318.734} C_VEL
LIN {X 0,Y 509.086,Z 520.01,A -85,B 0,C 180,E1 -5319.536,E2 -5319.536} C_VEL
LIN {X 0,Y 509.156,Z 520.052,A -85,B 0,C 180,E1 -5320.337,E2 -5320.337} C_VEL
LIN {X 0,Y 509.184,Z 519.435,A -85,B 0,C 180,E1 -5321.486,E2 -5321.486} C_VEL
LIN {X 0,Y 509.143,Z 517.766,A -85,B 0,C 180,E1 -5322.76,E2 -5322.76} C_VEL
LIN {X 0,Y 509.199,Z 515.174,A -85,B 0,C 180,E1 -5323.977,E2 -5323.977} C_VEL
LIN {X 0,Y 509.327,Z 511.52,A -85,B 0,C 180,E1 -5325.199,E2 -5325.199} C_VEL
LIN {X 0,Y 509.396,Z 506.676,A -85,B 0,C 180,E1 -5326.429,E2 -5326.429} C_VEL
LIN {X 0,Y 509.593,Z 500.49,A -85,B 0,C 180,E1 -5327.663,E2 -5327.663} C_VEL
LIN {X 0,Y 509.851,Z 492.719,A -85,B 0,C 180,E1 -5328.901,E2 -5328.901} C_VEL
LIN {X 0,Y 510.033,Z 484.657,A -85,B 0,C 180,E1 -5329.941,E2 -5329.941} C_VEL
LIN {X 0,Y 510.355,Z 474.704,A -85,B 0,C 180,E1 -5330.98,E2 -5330.98} C_VEL
LIN {X 0,Y 510.703,Z 463.542,A -85,B 0,C 180,E1 -5331.918,E2 -5331.918} C_VEL
LIN {X 0,Y 511.085,Z 452.526,A -85,B 0,C 180,E1 -5332.646,E2 -5332.646} C_VEL
LIN {X 0,Y 511.335,Z 439.814,A -85,B 0,C 180,E1 -5333.294,E2 -5333.294} C_VEL
LIN {X 0,Y 511.542,Z 426.697,A -85,B 0,C 180,E1 -5333.775,E2 -5333.775} C_VEL
LIN {X 0,Y 511.708,Z 414.442,A -85,B 0,C 180,E1 -5334.063,E2 -5334.063} C_VEL
LIN {X 0,Y 512.227,Z 320.349,A -85,B 0,C 180,E1 -5335.399,E2 -5335.399} C_VEL
LIN {X 0,Y 510.229,Z 309.39,A -85,B 0,C 180,E1 -5335.641,E2 -5335.641} C_VEL
LIN {X 0,Y 510.393,Z 294.121,A -85,B 0,C 180,E1 -5338.459,E2 -5338.459} C_VEL
LIN {X 0,Y 510.178,Z 288.546,A -85,B 0,C 180,E1 -5339.504,E2 -5339.504} C_VEL
LIN {X 0,Y 509.914,Z 286.973,A -85,B 0,C 180,E1 -5339.85,E2 -5339.85} C_VEL
LIN {X 0,Y 509.858,Z 286.972,A -85,B 0,C 180,E1 -5343.461,E2 -5343.461} C_VEL
LIN {X 0,Y 509.824,Z 286.982,A -85,B 0,C 180,E1 -5346.353,E2 -5346.353} C_VEL
LIN {X 0,Y 509.845,Z 286.973,A -85,B 0,C 180,E1 -5349.353,E2 -5349.353} C_VEL
LIN {X 0,Y 509.832,Z 286.98,A -85,B 0,C 180,E1 -5352.49,E2 -5352.49} C_VEL
LIN {X 0,Y 509.838,Z 286.974,A -85,B 0,C 180,E1 -5355.33,E2 -5355.33} C_VEL
LIN {X 0,Y 509.854,Z 286.977,A -85,B 0,C 180,E1 -5358.574,E2 -5358.574} C_VEL
LIN {X 0,Y 509.85,Z 286.969,A -85,B 0,C 180,E1 -5361.787,E2 -5361.787} C_VEL
LIN {X 0,Y 509.83,Z 286.976,A -85,B 0,C 180,E1 -5364.622,E2 -5364.622} C_VEL
LIN {X 0,Y 509.86,Z 286.97,A -85,B 0,C 180,E1 -5367.481,E2 -5367.481} C_VEL
LIN {X 0,Y 509.857,Z 286.967,A -85,B 0,C 180,E1 -5370.274,E2 -5370.274} C_VEL
LIN {X 0,Y 509.882,Z 286.969,A -85,B 0,C 180,E1 -5372.944,E2 -5372.944} C_VEL
LIN {X 0,Y 509.863,Z 286.97,A -85,B 0,C 180,E1 -5375.574,E2 -5375.574} C_VEL
LIN {X 0,Y 509.849,Z 286.973,A -85,B 0,C 180,E1 -5378.998,E2 -5378.998} C_VEL
LIN {X 0,Y 509.881,Z 286.969,A -85,B 0,C 180,E1 -5382.002,E2 -5382.002} C_VEL
LIN {X 0,Y 509.91,Z 286.961,A -85,B 0,C 180,E1 -5384.819,E2 -5384.819} C_VEL
LIN {X 0,Y 509.9,Z 286.965,A -85,B 0,C 180,E1 -5388.124,E2 -5388.124} C_VEL
LIN {X 0,Y 509.913,Z 286.965,A -85,B 0,C 180,E1 -5391.28,E2 -5391.28} C_VEL
LIN {X 0,Y 509.953,Z 286.963,A -85,B 0,C 180,E1 -5393.67,E2 -5393.67} C_VEL
LIN {X 0,Y 510.054,Z 286.948,A -85,B 0,C 180,E1 -5397.631,E2 -5397.631} C_VEL
LIN {X 0,Y 510.062,Z 286.944,A -85,B 0,C 180,E1 -5400.79,E2 -5400.79} C_VEL
LIN {X 0,Y 509.954,Z 286.955,A -85,B 0,C 180,E1 -5403.16,E2 -5403.16} C_VEL
LIN {X 0,Y 509.953,Z 286.962,A -85,B 0,C 180,E1 -5406.33,E2 -5406.33} C_VEL
LIN {X 0,Y 509.914,Z 286.965,A -85,B 0,C 180,E1 -5408.72,E2 -5408.72} C_VEL
LIN {X 0,Y 509.904,Z 286.963,A -85,B 0,C 180,E1 -5411.932,E2 -5411.932} C_VEL
LIN {X 0,Y 509.894,Z 286.963,A -85,B 0,C 180,E1 -5415.242,E2 -5415.242} C_VEL
LIN {X 0,Y 509.882,Z 286.967,A -85,B 0,C 180,E1 -5417.999,E2 -5417.999} C_VEL
LIN {X 0,Y 509.85,Z 286.974,A -85,B 0,C 180,E1 -5421.002,E2 -5421.002} C_VEL
LIN {X 0,Y 509.865,Z 286.972,A -85,B 0,C 180,E1 -5424.426,E2 -5424.426} C_VEL
LIN {X 0,Y 509.884,Z 286.972,A -85,B 0,C 180,E1 -5427.056,E2 -5427.056} C_VEL
LIN {X 0,Y 509.858,Z 286.97,A -85,B 0,C 180,E1 -5429.751,E2 -5429.751} C_VEL
LIN {X 0,Y 509.873,Z 286.972,A -85,B 0,C 180,E1 -5432.774,E2 -5432.774} C_VEL
LIN {X 0,Y 509.826,Z 286.975,A -85,B 0,C 180,E1 -5435.579,E2 -5435.579} C_VEL
LIN {X 0,Y 509.85,Z 286.97,A -85,B 0,C 180,E1 -5438.338,E2 -5438.338} C_VEL
LIN {X 0,Y 509.856,Z 286.973,A -85,B 0,C 180,E1 -5441.426,E2 -5441.426} C_VEL
LIN {X 0,Y 509.84,Z 286.971,A -85,B 0,C 180,E1 -5444.67,E2 -5444.67} C_VEL
LIN {X 0,Y 509.857,Z 286.972,A -85,B 0,C 180,E1 -5448.104,E2 -5448.104} C_VEL
LIN {X 0,Y 509.847,Z 286.971,A -85,B 0,C 180,E1 -5450.648,E2 -5450.648} C_VEL
LIN {X 0,Y 509.827,Z 286.98,A -85,B 0,C 180,E1 -5453.647,E2 -5453.647} C_VEL
LIN {X 0,Y 509.861,Z 286.971,A -85,B 0,C 180,E1 -5456.539,E2 -5456.539} C_VEL
LIN {X 0,Y 509.848,Z 286.975,A -85,B 0,C 180,E1 -5459.334,E2 -5459.334} C_VEL
LIN {X 0,Y 509.891,Z 286.972,A -85,B 0,C 180,E1 -5462.054,E2 -5462.054} C_VEL
LIN {X 0,Y 509.885,Z 286.972,A -85,B 0,C 180,E1 -5465.002,E2 -5465.002} C_VEL
LIN {X 0,Y 509.941,Z 287.25,A -85,B 0,C 180,E1 -5465.153,E2 -5465.153} C_VEL
LIN {X 0,Y 511.411,Z 295.127,A -85,B 0,C 180,E1 -5466.514,E2 -5466.514} C_VEL
LIN {X 0,Y 511.226,Z 306.973,A -85,B 0,C 180,E1 -5468.424,E2 -5468.424} C_VEL
LIN {X 0,Y 510.7,Z 326.713,A -85,B 0,C 180,E1 -5471.548,E2 -5471.548} C_VEL
LIN {X 0,Y 510.238,Z 345.071,A -85,B 0,C 180,E1 -5474.413,E2 -5474.413} C_VEL
LIN {X 0,Y 512.187,Z 358.672,A -85,B 0,C 180,E1 -5474.668,E2 -5474.668} C_VEL
LIN {X 0,Y 511.702,Z 453.321,A -85,B 0,C 180,E1 -5476.016,E2 -5476.016} C_VEL
LIN {X 0,Y 511.447,Z 466.662,A -85,B 0,C 180,E1 -5476.364,E2 -5476.364} C_VEL
LIN {X 0,Y 511.162,Z 478.868,A -85,B 0,C 180,E1 -5476.837,E2 -5476.837} C_VEL
LIN {X 0,Y 510.847,Z 491.44,A -85,B 0,C 180,E1 -5477.502,E2 -5477.502} C_VEL
LIN {X 0,Y 510.555,Z 502.816,A -85,B 0,C 180,E1 -5478.285,E2 -5478.285} C_VEL
LIN {X 0,Y 510.222,Z 513.286,A -85,B 0,C 180,E1 -5479.183,E2 -5479.183} C_VEL
LIN {X 0,Y 509.923,Z 521.848,A -85,B 0,C 180,E1 -5480.079,E2 -5480.079} C_VEL
LIN {X 0,Y 509.666,Z 529.75,A -85,B 0,C 180,E1 -5481.075,E2 -5481.075} C_VEL
LIN {X 0,Y 509.48,Z 537.47,A -85,B 0,C 180,E1 -5482.27,E2 -5482.27} C_VEL
LIN {X 0,Y 509.308,Z 544.585,A -85,B 0,C 180,E1 -5483.662,E2 -5483.662} C_VEL
LIN {X 0,Y 509.243,Z 549.321,A -85,B 0,C 180,E1 -5484.853,E2 -5484.853} C_VEL
LIN {X 0,Y 509.246,Z 552.942,A -85,B 0,C 180,E1 -5486.043,E2 -5486.043} C_VEL
LIN {X 0,Y 509.2,Z 554.808,A -85,B 0,C 180,E1 -5486.835,E2 -5486.835} C_VEL
LIN {X 0,Y 509.189,Z 556.208,A -85,B 0,C 180,E1 -5487.627,E2 -5487.627} C_VEL
LIN {X 0,Y 509.074,Z 557.815,A -85,B 0,C 180,E1 -5489.209,E2 -5489.209} C_VEL
LIN {X 0,Y 509.069,Z 558.033,A -85,B 0,C 180,E1 -5490,E2 -5490} C_VEL
LIN {X 0,Y 509.112,Z 557.212,A -85,B 0,C 180,E1 -5491.582,E2 -5491.582} C_VEL
LIN {X 0,Y 509.189,Z 556.219,A -85,B 0,C 180,E1 -5492.373,E2 -5492.373} C_VEL
LIN {X 0,Y 509.2,Z 554.822,A -85,B 0,C 180,E1 -5493.164,E2 -5493.164} C_VEL
LIN {X 0,Y 509.204,Z 551.882,A -85,B 0,C 180,E1 -5494.353,E2 -5494.353} C_VEL
LIN {X 0,Y 509.292,Z 547.904,A -85,B 0,C 180,E1 -5495.543,E2 -5495.543} C_VEL
LIN {X 0,Y 509.372,Z 542.237,A -85,B 0,C 180,E1 -5496.844,E2 -5496.844} C_VEL
LIN {X 0,Y 509.544,Z 535.094,A -85,B 0,C 180,E1 -5498.127,E2 -5498.127} C_VEL
LIN {X 0,Y 509.756,Z 526.796,A -85,B 0,C 180,E1 -5499.322,E2 -5499.322} C_VEL
LIN {X 0,Y 510.012,Z 518.291,A -85,B 0,C 180,E1 -5500.319,E2 -5500.319} C_VEL
LIN {X 0,Y 510.389,Z 507.786,A -85,B 0,C 180,E1 -5501.316,E2 -5501.316} C_VEL
LIN {X 0,Y 510.709,Z 496.318,A -85,B 0,C 180,E1 -5502.189,E2 -5502.189} C_VEL
LIN {X 0,Y 511.007,Z 486.001,A -85,B 0,C 180,E1 -5502.813,E2 -5502.813} C_VEL
LIN {X 0,Y 511.297,Z 474.307,A -85,B 0,C 180,E1 -5503.361,E2 -5503.361} C_VEL
LIN {X 0,Y 511.556,Z 460.834,A -85,B 0,C 180,E1 -5503.81,E2 -5503.81} C_VEL
LIN {X 0,Y 511.793,Z 447.49,A -85,B 0,C 180,E1 -5504.082,E2 -5504.082} C_VEL
LIN {X 0,Y 512.149,Z 357.844,A -85,B 0,C 180,E1 -5505.346,E2 -5505.346} C_VEL
LIN {X 0,Y 510.247,Z 345.144,A -85,B 0,C 180,E1 -5505.588,E2 -5505.588} C_VEL
LIN {X 0,Y 510.742,Z 325.559,A -85,B 0,C 180,E1 -5508.658,E2 -5508.658} C_VEL
LIN {X 0,Y 511.243,Z 307.172,A -85,B 0,C 180,E1 -5511.575,E2 -5511.575} C_VEL
LIN {X 0,Y 511.587,Z 297.183,A -85,B 0,C 180,E1 -5513.173,E2 -5513.173} C_VEL
LIN {X 0,Y 510.498,Z 289.962,A -85,B 0,C 180,E1 -5514.393,E2 -5514.393} C_VEL
LIN {X 0,Y 509.906,Z 286.97,A -85,B 0,C 180,E1 -5514.95,E2 -5514.95} C_VEL
LIN {X 0,Y 509.894,Z 286.974,A -85,B 0,C 180,E1 -5517.945,E2 -5517.945} C_VEL
LIN {X 0,Y 509.845,Z 286.972,A -85,B 0,C 180,E1 -5520.665,E2 -5520.665} C_VEL
LIN {X 0,Y 509.859,Z 286.97,A -85,B 0,C 180,E1 -5523.46,E2 -5523.46} C_VEL
LIN {X 0,Y 509.824,Z 286.982,A -85,B 0,C 180,E1 -5526.352,E2 -5526.352} C_VEL
LIN {X 0,Y 509.844,Z 286.971,A -85,B 0,C 180,E1 -5529.352,E2 -5529.352} C_VEL
LIN {X 0,Y 509.832,Z 286.981,A -85,B 0,C 180,E1 -5532.489,E2 -5532.489} C_VEL
LIN {X 0,Y 509.836,Z 286.972,A -85,B 0,C 180,E1 -5535.329,E2 -5535.329} C_VEL
LIN {X 0,Y 509.855,Z 286.979,A -85,B 0,C 180,E1 -5538.574,E2 -5538.574} C_VEL
LIN {X 0,Y 509.848,Z 286.97,A -85,B 0,C 180,E1 -5541.786,E2 -5541.786} C_VEL
LIN {X 0,Y 509.828,Z 286.98,A -85,B 0,C 180,E1 -5544.621,E2 -5544.621} C_VEL
LIN {X 0,Y 509.858,Z 286.97,A -85,B 0,C 180,E1 -5547.48,E2 -5547.48} C_VEL
LIN {X 0,Y 509.855,Z 286.971,A -85,B 0,C 180,E1 -5550.273,E2 -5550.273} C_VEL
LIN {X 0,Y 509.881,Z 286.975,A -85,B 0,C 180,E1 -5552.944,E2 -5552.944} C_VEL
LIN {X 0,Y 509.866,Z 286.97,A -85,B 0,C 180,E1 -5555.574,E2 -5555.574} C_VEL
LIN {X 0,Y 509.846,Z 286.978,A -85,B 0,C 180,E1 -5558.998,E2 -5558.998} C_VEL
LIN {X 0,Y 509.884,Z 286.966,A -85,B 0,C 180,E1 -5561.999,E2 -5561.999} C_VEL
LIN {X 0,Y 509.906,Z 286.966,A -85,B 0,C 180,E1 -5564.818,E2 -5564.818} C_VEL
LIN {X 0,Y 509.896,Z 286.965,A -85,B 0,C 180,E1 -5568.124,E2 -5568.124} C_VEL
LIN {X 0,Y 509.911,Z 286.969,A -85,B 0,C 180,E1 -5571.28,E2 -5571.28} C_VEL
LIN {X 0,Y 509.966,Z 286.963,A -85,B 0,C 180,E1 -5573.67,E2 -5573.67} C_VEL
LIN {X 0,Y 510.048,Z 286.955,A -85,B 0,C 180,E1 -5577.631,E2 -5577.631} C_VEL
LIN {X 0,Y 510.049,Z 286.95,A -85,B 0,C 180,E1 -5580,E2 -5580} C_VEL
LIN {X 0,Y 510.048,Z 286.947,A -85,B 0,C 180,E1 -5582.369,E2 -5582.369} C_VEL
LIN {X 0,Y 509.97,Z 286.959,A -85,B 0,C 180,E1 -5585.536,E2 -5585.536} C_VEL
LIN {X 0,Y 509.909,Z 286.963,A -85,B 0,C 180,E1 -5588.72,E2 -5588.72} C_VEL
LIN {X 0,Y 509.898,Z 286.972,A -85,B 0,C 180,E1 -5591.932,E2 -5591.932} C_VEL
LIN {X 0,Y 509.888,Z 286.965,A -85,B 0,C 180,E1 -5595.242,E2 -5595.242} C_VEL
LIN {X 0,Y 509.855,Z 286.975,A -85,B 0,C 180,E1 -5598.484,E2 -5598.484} C_VEL
LIN {X 0,Y 509.844,Z 286.972,A -85,B 0,C 180,E1 -5601.002,E2 -5601.002} C_VEL
LIN {X 0,Y 509.816,Z 286.974,A -85,B 0,C 180,E1 -5603.564,E2 -5603.564} C_VEL
LIN {X 0,Y 509.902,Z 286.972,A -85,B 0,C 180,E1 -5606.378,E2 -5606.378} C_VEL
LIN {X 0,Y 509.866,Z 286.972,A -85,B 0,C 180,E1 -5608.845,E2 -5608.845} C_VEL
LIN {X 0,Y 509.814,Z 286.974,A -85,B 0,C 180,E1 -5611.59,E2 -5611.59} C_VEL
LIN {X 0,Y 509.842,Z 286.977,A -85,B 0,C 180,E1 -5614.414,E2 -5614.414} C_VEL
LIN {X 0,Y 509.811,Z 286.976,A -85,B 0,C 180,E1 -5617.341,E2 -5617.341} C_VEL
LIN {X 0,Y 509.832,Z 286.975,A -85,B 0,C 180,E1 -5620.383,E2 -5620.383} C_VEL
LIN {X 0,Y 509.818,Z 286.981,A -85,B 0,C 180,E1 -5623.062,E2 -5623.062} C_VEL
LIN {X 0,Y 509.825,Z 286.973,A -85,B 0,C 180,E1 -5625.793,E2 -5625.793} C_VEL
LIN {X 0,Y 509.827,Z 286.975,A -85,B 0,C 180,E1 -5628.573,E2 -5628.573} C_VEL
LIN {X 0,Y 509.845,Z 286.972,A -85,B 0,C 180,E1 -5631.787,E2 -5631.787} C_VEL
LIN {X 0,Y 509.817,Z 286.976,A -85,B 0,C 180,E1 -5633.718,E2 -5633.718} C_VEL
LIN {X 0,Y 509.148,Z 287.058,A -85,B 0,C 180,E1 -5634.377,E2 -5634.377} C_VEL
LIN {X 0,Y 506.336,Z 287.414,A -85,B 0,C 180,E1 -5635.449,E2 -5635.449} C_VEL
LIN {X 0,Y 503.95,Z 287.712,A -85,B 0,C 180,E1 -5636.313,E2 -5636.313} C_VEL
LIN {X 0,Y 502.903,Z 287.84,A -85,B 0,C 180,E1 -5636.979,E2 -5636.979} C_VEL
LIN {X 0,Y 502.804,Z 287.85,A -85,B 0,C 180,E1 -5637.205,E2 -5637.205} C_VEL
LIN {X 0,Y 502.808,Z 287.848,A -85,B 0,C 180,E1 -5640.066,E2 -5640.066} C_VEL
LIN {X 0,Y 502.78,Z 287.86,A -85,B 0,C 180,E1 -5643.43,E2 -5643.43} C_VEL
LIN {X 0,Y 502.764,Z 287.855,A -85,B 0,C 180,E1 -5646.085,E2 -5646.085} C_VEL
LIN {X 0,Y 502.781,Z 287.851,A -85,B 0,C 180,E1 -5648.689,E2 -5648.689} C_VEL
LIN {X 0,Y 502.81,Z 287.85,A -85,B 0,C 180,E1 -5651.248,E2 -5651.248} C_VEL
LIN {X 0,Y 502.837,Z 287.844,A -85,B 0,C 180,E1 -5654.664,E2 -5654.664} C_VEL
LIN {X 0,Y 502.868,Z 287.849,A -85,B 0,C 180,E1 -5658.044,E2 -5658.044} C_VEL
LIN {X 0,Y 502.834,Z 287.925,A -85,B 0,C 180,E1 -5660.04,E2 -5660.04} C_VEL
LIN {X 0,Y 503.485,Z 292.566,A -85,B 0,C 180,E1 -5660.966,E2 -5660.966} C_VEL
LIN {X 0,Y 503.256,Z 307.334,A -85,B 0,C 180,E1 -5663.787,E2 -5663.787} C_VEL
LIN {X 0,Y 503.21,Z 309.724,A -85,B 0,C 180,E1 -5664.239,E2 -5664.239} C_VEL
LIN {X 0,Y 505.38,Z 321.277,A -85,B 0,C 180,E1 -5664.489,E2 -5664.489} C_VEL
LIN {X 0,Y 504.847,Z 417.286,A -85,B 0,C 180,E1 -5665.884,E2 -5665.884} C_VEL
LIN {X 0,Y 504.639,Z 430.917,A -85,B 0,C 180,E1 -5666.257,E2 -5666.257} C_VEL
LIN {X 0,Y 504.428,Z 443.159,A -85,B 0,C 180,E1 -5666.756,E2 -5666.756} C_VEL
LIN {X 0,Y 504.09,Z 454.935,A -85,B 0,C 180,E1 -5667.403,E2 -5667.403} C_VEL
LIN {X 0,Y 503.646,Z 466.247,A -85,B 0,C 180,E1 -5668.201,E2 -5668.201} C_VEL
LIN {X 0,Y 503.249,Z 476.451,A -85,B 0,C 180,E1 -5669.1,E2 -5669.1} C_VEL
LIN {X 0,Y 503.081,Z 484.78,A -85,B 0,C 180,E1 -5670,E2 -5670} C_VEL
LIN {X 0,Y 502.779,Z 492.518,A -85,B 0,C 180,E1 -5671.001,E2 -5671.001} C_VEL
LIN {X 0,Y 502.509,Z 500.096,A -85,B 0,C 180,E1 -5672.204,E2 -5672.204} C_VEL
LIN {X 0,Y 502.341,Z 507.088,A -85,B 0,C 180,E1 -5673.61,E2 -5673.61} C_VEL
LIN {X 0,Y 502.158,Z 511.766,A -85,B 0,C 180,E1 -5674.817,E2 -5674.817} C_VEL
LIN {X 0,Y 502.175,Z 515.824,A -85,B 0,C 180,E1 -5676.213,E2 -5676.213} C_VEL
LIN {X 0,Y 502.111,Z 517.922,A -85,B 0,C 180,E1 -5677.237,E2 -5677.237} C_VEL
LIN {X 0,Y 502.09,Z 519.14,A -85,B 0,C 180,E1 -5678.047,E2 -5678.047} C_VEL
LIN {X 0,Y 502.038,Z 519.926,A -85,B 0,C 180,E1 -5678.858,E2 -5678.858} C_VEL
LIN {X 0,Y 502.062,Z 520.289,A -85,B 0,C 180,E1 -5680.485,E2 -5680.485} C_VEL
LIN {X 0,Y 502.103,Z 519.669,A -85,B 0,C 180,E1 -5681.537,E2 -5681.537} C_VEL
LIN {X 0,Y 502.047,Z 517.772,A -85,B 0,C 180,E1 -5682.943,E2 -5682.943} C_VEL
LIN {X 0,Y 502.146,Z 515.058,A -85,B 0,C 180,E1 -5684.178,E2 -5684.178} C_VEL
LIN {X 0,Y 502.244,Z 511.271,A -85,B 0,C 180,E1 -5685.419,E2 -5685.419} C_VEL
LIN {X 0,Y 502.355,Z 506.287,A -85,B 0,C 180,E1 -5686.666,E2 -5686.666} C_VEL
LIN {X 0,Y 502.619,Z 499.233,A -85,B 0,C 180,E1 -5688.043,E2 -5688.043} C_VEL
LIN {X 0,Y 502.815,Z 491.917,A -85,B 0,C 180,E1 -5689.176,E2 -5689.176} C_VEL
LIN {X 0,Y 503.084,Z 483.619,A -85,B 0,C 180,E1 -5690.228,E2 -5690.228} C_VEL
LIN {X 0,Y 503.464,Z 473.405,A -85,B 0,C 180,E1 -5691.281,E2 -5691.281} C_VEL
LIN {X 0,Y 503.786,Z 463.229,A -85,B 0,C 180,E1 -5692.127,E2 -5692.127} C_VEL
LIN {X 0,Y 504.187,Z 452.031,A -85,B 0,C 180,E1 -5692.865,E2 -5692.865} C_VEL
LIN {X 0,Y 504.433,Z 440.129,A -85,B 0,C 180,E1 -5693.476,E2 -5693.476} C_VEL
LIN {X 0,Y 504.659,Z 427.285,A -85,B 0,C 180,E1 -5693.956,E2 -5693.956} C_VEL
LIN {X 0,Y 504.829,Z 415.264,A -85,B 0,C 180,E1 -5694.248,E2 -5694.248} C_VEL
LIN {X 0,Y 505.398,Z 321.132,A -85,B 0,C 180,E1 -5695.605,E2 -5695.605} C_VEL
LIN {X 0,Y 503.249,Z 309.652,A -85,B 0,C 180,E1 -5695.855,E2 -5695.855} C_VEL
LIN {X 0,Y 503.45,Z 292.786,A -85,B 0,C 180,E1 -5698.996,E2 -5698.996} C_VEL
LIN {X 0,Y 502.872,Z 287.85,A -85,B 0,C 180,E1 -5699.992,E2 -5699.992} C_VEL
LIN {X 0,Y 502.831,Z 287.848,A -85,B 0,C 180,E1 -5703.031,E2 -5703.031} C_VEL
LIN {X 0,Y 502.773,Z 287.857,A -85,B 0,C 180,E1 -5705.951,E2 -5705.951} C_VEL
LIN {X 0,Y 502.8,Z 287.853,A -85,B 0,C 180,E1 -5708.976,E2 -5708.976} C_VEL
LIN {X 0,Y 502.794,Z 287.854,A -85,B 0,C 180,E1 -5712.139,E2 -5712.139} C_VEL
LIN {X 0,Y 502.784,Z 287.852,A -85,B 0,C 180,E1 -5715.47,E2 -5715.47} C_VEL
LIN {X 0,Y 502.819,Z 287.853,A -85,B 0,C 180,E1 -5718.934,E2 -5718.934} C_VEL
LIN {X 0,Y 502.792,Z 287.849,A -85,B 0,C 180,E1 -5722.046,E2 -5722.046} C_VEL
LIN {X 0,Y 502.799,Z 287.856,A -85,B 0,C 180,E1 -5725.034,E2 -5725.034} C_VEL
LIN {X 0,Y 502.782,Z 287.849,A -85,B 0,C 180,E1 -5727.915,E2 -5727.915} C_VEL
LIN {X 0,Y 502.823,Z 287.847,A -85,B 0,C 180,E1 -5730.712,E2 -5730.712} C_VEL
LIN {X 0,Y 502.862,Z 287.845,A -85,B 0,C 180,E1 -5733.439,E2 -5733.439} C_VEL
LIN {X 0,Y 502.784,Z 287.847,A -85,B 0,C 180,E1 -5736.086,E2 -5736.086} C_VEL
LIN {X 0,Y 502.782,Z 287.851,A -85,B 0,C 180,E1 -5738.689,E2 -5738.689} C_VEL
LIN {X 0,Y 502.828,Z 287.848,A -85,B 0,C 180,E1 -5741.248,E2 -5741.248} C_VEL
LIN {X 0,Y 502.821,Z 287.849,A -85,B 0,C 180,E1 -5743.767,E2 -5743.767} C_VEL
LIN {X 0,Y 502.829,Z 287.846,A -85,B 0,C 180,E1 -5746.255,E2 -5746.255} C_VEL
LIN {X 0,Y 502.876,Z 287.837,A -85,B 0,C 180,E1 -5748.717,E2 -5748.717} C_VEL
LIN {X 0,Y 502.901,Z 287.841,A -85,B 0,C 180,E1 -5751.967,E2 -5751.967} C_VEL
LIN {X 0,Y 502.931,Z 287.834,A -85,B 0,C 180,E1 -5754.387,E2 -5754.387} C_VEL
LIN {X 0,Y 503.024,Z 287.824,A -85,B 0,C 180,E1 -5757.598,E2 -5757.598} C_VEL
LIN {X 0,Y 503.027,Z 287.828,A -85,B 0,C 180,E1 -5760,E2 -5760} C_VEL
LIN {X 0,Y 503.023,Z 287.823,A -85,B 0,C 180,E1 -5762.402,E2 -5762.402} C_VEL
LIN {X 0,Y 502.931,Z 287.833,A -85,B 0,C 180,E1 -5765.614,E2 -5765.614} C_VEL
LIN {X 0,Y 502.901,Z 287.838,A -85,B 0,C 180,E1 -5768.034,E2 -5768.034} C_VEL
LIN {X 0,Y 502.876,Z 287.836,A -85,B 0,C 180,E1 -5771.283,E2 -5771.283} C_VEL
LIN {X 0,Y 502.845,Z 287.849,A -85,B 0,C 180,E1 -5774.571,E2 -5774.571} C_VEL
LIN {X 0,Y 502.855,Z 287.842,A -85,B 0,C 180,E1 -5777.907,E2 -5777.907} C_VEL
LIN {X 0,Y 502.829,Z 287.85,A -85,B 0,C 180,E1 -5780.536,E2 -5780.536} C_VEL
LIN {X 0,Y 502.791,Z 287.854,A -85,B 0,C 180,E1 -5783.041,E2 -5783.041} C_VEL
LIN {X 0,Y 502.84,Z 287.843,A -85,B 0,C 180,E1 -5785.676,E2 -5785.676} C_VEL
LIN {X 0,Y 502.84,Z 287.845,A -85,B 0,C 180,E1 -5788.373,E2 -5788.373} C_VEL
LIN {X 0,Y 502.793,Z 287.851,A -85,B 0,C 180,E1 -5791.499,E2 -5791.499} C_VEL
LIN {X 0,Y 502.804,Z 287.848,A -85,B 0,C 180,E1 -5793.994,E2 -5793.994} C_VEL
LIN {X 0,Y 502.778,Z 287.859,A -85,B 0,C 180,E1 -5797.178,E2 -5797.178} C_VEL
LIN {X 0,Y 502.788,Z 287.843,A -85,B 0,C 180,E1 -5800.015,E2 -5800.015} C_VEL
LIN {X 0,Y 502.804,Z 287.848,A -85,B 0,C 180,E1 -5802.199,E2 -5802.199} C_VEL
LIN {X 0,Y 502.787,Z 287.86,A -85,B 0,C 180,E1 -5805.47,E2 -5805.47} C_VEL
LIN {X 0,Y 502.821,Z 287.848,A -85,B 0,C 180,E1 -5808.934,E2 -5808.934} C_VEL
LIN {X 0,Y 502.795,Z 287.851,A -85,B 0,C 180,E1 -5812.046,E2 -5812.046} C_VEL
LIN {X 0,Y 502.801,Z 287.851,A -85,B 0,C 180,E1 -5815.034,E2 -5815.034} C_VEL
LIN {X 0,Y 502.785,Z 287.858,A -85,B 0,C 180,E1 -5817.916,E2 -5817.916} C_VEL
LIN {X 0,Y 502.826,Z 287.848,A -85,B 0,C 180,E1 -5820.712,E2 -5820.712} C_VEL
LIN {X 0,Y 502.866,Z 287.845,A -85,B 0,C 180,E1 -5823.439,E2 -5823.439} C_VEL
LIN {X 0,Y 502.87,Z 287.924,A -85,B 0,C 180,E1 -5824.922,E2 -5824.922} C_VEL
LIN {X 0,Y 504.523,Z 297.279,A -85,B 0,C 180,E1 -5826.562,E2 -5826.562} C_VEL
LIN {X 0,Y 504.146,Z 312.085,A -85,B 0,C 180,E1 -5828.975,E2 -5828.975} C_VEL
LIN {X 0,Y 503.588,Z 331.711,A -85,B 0,C 180,E1 -5832.12,E2 -5832.12} C_VEL
LIN {X 0,Y 503.235,Z 344.894,A -85,B 0,C 180,E1 -5834.192,E2 -5834.192} C_VEL
LIN {X 0,Y 505.347,Z 359.672,A -85,B 0,C 180,E1 -5834.473,E2 -5834.473} C_VEL
LIN {X 0,Y 504.831,Z 453.024,A -85,B 0,C 180,E1 -5835.822,E2 -5835.822} C_VEL
LIN {X 0,Y 504.581,Z 465.611,A -85,B 0,C 180,E1 -5836.149,E2 -5836.149} C_VEL
LIN {X 0,Y 504.243,Z 478.584,A -85,B 0,C 180,E1 -5836.653,E2 -5836.653} C_VEL
LIN {X 0,Y 503.905,Z 490.554,A -85,B 0,C 180,E1 -5837.288,E2 -5837.288} C_VEL
LIN {X 0,Y 503.567,Z 502.537,A -85,B 0,C 180,E1 -5838.12,E2 -5838.12} C_VEL
LIN {X 0,Y 503.22,Z 513.01,A -85,B 0,C 180,E1 -5839.03,E2 -5839.03} C_VEL
LIN {X 0,Y 502.873,Z 521.572,A -85,B 0,C 180,E1 -5839.939,E2 -5839.939} C_VEL
LIN {X 0,Y 502.621,Z 529.476,A -85,B 0,C 180,E1 -5840.949,E2 -5840.949} C_VEL
LIN {X 0,Y 502.4,Z 537.198,A -85,B 0,C 180,E1 -5842.161,E2 -5842.161} C_VEL
LIN {X 0,Y 502.236,Z 544.316,A -85,B 0,C 180,E1 -5843.572,E2 -5843.572} C_VEL
LIN {X 0,Y 502.175,Z 549.054,A -85,B 0,C 180,E1 -5844.78,E2 -5844.78} C_VEL
LIN {X 0,Y 502.139,Z 552.674,A -85,B 0,C 180,E1 -5845.987,E2 -5845.987} C_VEL
LIN {X 0,Y 502.12,Z 554.542,A -85,B 0,C 180,E1 -5846.79,E2 -5846.79} C_VEL
LIN {X 0,Y 502.091,Z 555.943,A -85,B 0,C 180,E1 -5847.593,E2 -5847.593} C_VEL
LIN {X 0,Y 501.99,Z 557.551,A -85,B 0,C 180,E1 -5849.198,E2 -5849.198} C_VEL
LIN {X 0,Y 501.983,Z 557.769,A -85,B 0,C 180,E1 -5850,E2 -5850} C_VEL
LIN {X 0,Y 502.036,Z 556.949,A -85,B 0,C 180,E1 -5851.604,E2 -5851.604} C_VEL
LIN {X 0,Y 502.091,Z 555.956,A -85,B 0,C 180,E1 -5852.406,E2 -5852.406} C_VEL
LIN {X 0,Y 502.12,Z 554.559,A -85,B 0,C 180,E1 -5853.209,E2 -5853.209} C_VEL
LIN {X 0,Y 502.102,Z 551.618,A -85,B 0,C 180,E1 -5854.415,E2 -5854.415} C_VEL
LIN {X 0,Y 502.208,Z 547.639,A -85,B 0,C 180,E1 -5855.621,E2 -5855.621} C_VEL
LIN {X 0,Y 502.324,Z 541.619,A -85,B 0,C 180,E1 -5857.011,E2 -5857.011} C_VEL
LIN {X 0,Y 502.477,Z 534.828,A -85,B 0,C 180,E1 -5858.242,E2 -5858.242} C_VEL
LIN {X 0,Y 502.716,Z 526.529,A -85,B 0,C 180,E1 -5859.454,E2 -5859.454} C_VEL
LIN {X 0,Y 502.989,Z 518.023,A -85,B 0,C 180,E1 -5860.465,E2 -5860.465} C_VEL
LIN {X 0,Y 503.406,Z 507.518,A -85,B 0,C 180,E1 -5861.475,E2 -5861.475} C_VEL
LIN {X 0,Y 503.737,Z 496.048,A -85,B 0,C 180,E1 -5862.361,E2 -5862.361} C_VEL
LIN {X 0,Y 504.06,Z 485.728,A -85,B 0,C 180,E1 -5862.992,E2 -5862.992} C_VEL
LIN {X 0,Y 504.396,Z 474.031,A -85,B 0,C 180,E1 -5863.547,E2 -5863.547} C_VEL
LIN {X 0,Y 504.677,Z 460.553,A -85,B 0,C 180,E1 -5864.002,E2 -5864.002} C_VEL
LIN {X 0,Y 504.926,Z 447.193,A -85,B 0,C 180,E1 -5864.277,E2 -5864.277} C_VEL
LIN {X 0,Y 505.311,Z 358.884,A -85,B 0,C 180,E1 -5865.54,E2 -5865.54} C_VEL
LIN {X 0,Y 503.244,Z 344.821,A -85,B 0,C 180,E1 -5865.82,E2 -5865.82} C_VEL
LIN {X 0,Y 503.765,Z 325.28,A -85,B 0,C 180,E1 -5868.926,E2 -5868.926} C_VEL
LIN {X 0,Y 504.286,Z 308.179,A -85,B 0,C 180,E1 -5871.673,E2 -5871.673} C_VEL
LIN {X 0,Y 504.558,Z 297.265,A -85,B 0,C 180,E1 -5873.447,E2 -5873.447} C_VEL
LIN {X 0,Y 502.873,Z 287.846,A -85,B 0,C 180,E1 -5875.108,E2 -5875.108} C_VEL
LIN {X 0,Y 502.845,Z 287.851,A -85,B 0,C 180,E1 -5878.295,E2 -5878.295} C_VEL
LIN {X 0,Y 502.793,Z 287.85,A -85,B 0,C 180,E1 -5881.498,E2 -5881.498} C_VEL
LIN {X 0,Y 502.803,Z 287.854,A -85,B 0,C 180,E1 -5883.993,E2 -5883.993} C_VEL
LIN {X 0,Y 502.776,Z 287.851,A -85,B 0,C 180,E1 -5887.177,E2 -5887.177} C_VEL
LIN {X 0,Y 502.786,Z 287.854,A -85,B 0,C 180,E1 -5890.015,E2 -5890.015} C_VEL
LIN {X 0,Y 502.801,Z 287.854,A -85,B 0,C 180,E1 -5892.199,E2 -5892.199} C_VEL
LIN {X 0,Y 502.783,Z 287.85,A -85,B 0,C 180,E1 -5895.469,E2 -5895.469} C_VEL
LIN {X 0,Y 502.818,Z 287.85,A -85,B 0,C 180,E1 -5898.934,E2 -5898.934} C_VEL
LIN {X 0,Y 502.79,Z 287.851,A -85,B 0,C 180,E1 -5902.045,E2 -5902.045} C_VEL
LIN {X 0,Y 502.796,Z 287.854,A -85,B 0,C 180,E1 -5905.034,E2 -5905.034} C_VEL
LIN {X 0,Y 502.78,Z 287.851,A -85,B 0,C 180,E1 -5907.915,E2 -5907.915} C_VEL
LIN {X 0,Y 502.82,Z 287.852,A -85,B 0,C 180,E1 -5910.712,E2 -5910.712} C_VEL
LIN {X 0,Y 502.859,Z 287.844,A -85,B 0,C 180,E1 -5913.439,E2 -5913.439} C_VEL
LIN {X 0,Y 502.788,Z 287.85,A -85,B 0,C 180,E1 -5916.086,E2 -5916.086} C_VEL
LIN {X 0,Y 502.779,Z 287.854,A -85,B 0,C 180,E1 -5918.688,E2 -5918.688} C_VEL
LIN {X 0,Y 502.825,Z 287.854,A -85,B 0,C 180,E1 -5921.248,E2 -5921.248} C_VEL
LIN {X 0,Y 502.817,Z 287.849,A -85,B 0,C 180,E1 -5923.767,E2 -5923.767} C_VEL
LIN {X 0,Y 502.83,Z 287.844,A -85,B 0,C 180,E1 -5926.254,E2 -5926.254} C_VEL
LIN {X 0,Y 502.872,Z 287.84,A -85,B 0,C 180,E1 -5928.717,E2 -5928.717} C_VEL
LIN {X 0,Y 502.897,Z 287.839,A -85,B 0,C 180,E1 -5931.966,E2 -5931.966} C_VEL
LIN {X 0,Y 502.93,Z 287.832,A -85,B 0,C 180,E1 -5934.386,E2 -5934.386} C_VEL
LIN {X 0,Y 503.018,Z 287.83,A -85,B 0,C 180,E1 -5937.598,E2 -5937.598} C_VEL
LIN {X 0,Y 503.02,Z 287.826,A -85,B 0,C 180,E1 -5940,E2 -5940} C_VEL
LIN {X 0,Y 503.018,Z 287.823,A -85,B 0,C 180,E1 -5942.402,E2 -5942.402} C_VEL
LIN {X 0,Y 502.922,Z 287.838,A -85,B 0,C 180,E1 -5945.613,E2 -5945.613} C_VEL
LIN {X 0,Y 502.867,Z 287.84,A -85,B 0,C 180,E1 -5948.843,E2 -5948.843} C_VEL
LIN {X 0,Y 502.84,Z 287.852,A -85,B 0,C 180,E1 -5952.102,E2 -5952.102} C_VEL
LIN {X 0,Y 502.843,Z 287.843,A -85,B 0,C 180,E1 -5955.4,E2 -5955.4} C_VEL
LIN {X 0,Y 502.82,Z 287.848,A -85,B 0,C 180,E1 -5958.752,E2 -5958.752} C_VEL
LIN {X 0,Y 502.777,Z 287.851,A -85,B 0,C 180,E1 -5961.311,E2 -5961.311} C_VEL
LIN {X 0,Y 502.769,Z 287.855,A -85,B 0,C 180,E1 -5963.915,E2 -5963.915} C_VEL
LIN {X 0,Y 502.841,Z 287.851,A -85,B 0,C 180,E1 -5966.567,E2 -5966.567} C_VEL
LIN {X 0,Y 502.816,Z 287.847,A -85,B 0,C 180,E1 -5969.288,E2 -5969.288} C_VEL
LIN {X 0,Y 502.777,Z 287.853,A -85,B 0,C 180,E1 -5972.085,E2 -5972.085} C_VEL
LIN {X 0,Y 502.793,Z 287.854,A -85,B 0,C 180,E1 -5974.966,E2 -5974.966} C_VEL
LIN {X 0,Y 502.787,Z 287.85,A -85,B 0,C 180,E1 -5977.954,E2 -5977.954} C_VEL
LIN {X 0,Y 502.815,Z 287.852,A -85,B 0,C 180,E1 -5981.066,E2 -5981.066} C_VEL
LIN {X 0,Y 502.796,Z 287.852,A -85,B 0,C 180,E1 -5984.532,E2 -5984.532} C_VEL
LIN {X 0,Y 502.79,Z 287.85,A -85,B 0,C 180,E1 -5987.861,E2 -5987.861} C_VEL
LIN {X 0,Y 502.789,Z 287.858,A -85,B 0,C 180,E1 -5991.024,E2 -5991.024} C_VEL
LIN {X 0,Y 502.771,Z 287.852,A -85,B 0,C 180,E1 -5994.17,E2 -5994.17} C_VEL
LIN {X 0,Y 502.804,Z 287.85,A -85,B 0,C 180,E1 -5997.205,E2 -5997.205} C_VEL
LIN {X 0,Y 502.103,Z 287.938,A -85,B 0,C 180,E1 -5997.873,E2 -5997.873} C_VEL
LIN {X 0,Y 499.242,Z 288.295,A -85,B 0,C 180,E1 -5998.959,E2 -5998.959} C_VEL
LIN {X 0,Y 496.843,Z 288.593,A -85,B 0,C 180,E1 -5999.834,E2 -5999.834} C_VEL
LIN {X 0,Y 495.812,Z 288.719,A -85,B 0,C 180,E1 -6000.509,E2 -6000.509} C_VEL
LIN {X 0,Y 495.726,Z 288.731,A -85,B 0,C 180,E1 -6000.738,E2 -6000.738} C_VEL
LIN {X 0,Y 495.713,Z 288.734,A -85,B 0,C 180,E1 -6003.928,E2 -6003.928} C_VEL
LIN {X 0,Y 495.756,Z 288.729,A -85,B 0,C 180,E1 -6007.14,E2 -6007.14} C_VEL
LIN {X 0,Y 495.766,Z 288.727,A -85,B 0,C 180,E1 -6010.11,E2 -6010.11} C_VEL
LIN {X 0,Y 495.743,Z 288.727,A -85,B 0,C 180,E1 -6012.68,E2 -6012.68} C_VEL
LIN {X 0,Y 495.786,Z 288.724,A -85,B 0,C 180,E1 -6015.217,E2 -6015.217} C_VEL
LIN {X 0,Y 495.82,Z 288.723,A -85,B 0,C 180,E1 -6018.554,E2 -6018.554} C_VEL
LIN {X 0,Y 495.769,Z 288.841,A -85,B 0,C 180,E1 -6019.923,E2 -6019.923} C_VEL
LIN {X 0,Y 496.486,Z 294.447,A -85,B 0,C 180,E1 -6021.042,E2 -6021.042} C_VEL
LIN {X 0,Y 496.272,Z 308.267,A -85,B 0,C 180,E1 -6023.699,E2 -6023.699} C_VEL
LIN {X 0,Y 496.225,Z 309.961,A -85,B 0,C 180,E1 -6024.021,E2 -6024.021} C_VEL
LIN {X 0,Y 498.587,Z 322.342,A -85,B 0,C 180,E1 -6024.287,E2 -6024.287} C_VEL
LIN {X 0,Y 498.011,Z 417.001,A -85,B 0,C 180,E1 -6025.675,E2 -6025.675} C_VEL
LIN {X 0,Y 497.769,Z 430.091,A -85,B 0,C 180,E1 -6026.028,E2 -6026.028} C_VEL
LIN {X 0,Y 497.536,Z 443.175,A -85,B 0,C 180,E1 -6026.559,E2 -6026.559} C_VEL
LIN {X 0,Y 497.198,Z 454.248,A -85,B 0,C 180,E1 -6027.165,E2 -6027.165} C_VEL
LIN {X 0,Y 496.716,Z 465.742,A -85,B 0,C 180,E1 -6027.973,E2 -6027.973} C_VEL
LIN {X 0,Y 496.323,Z 476.074,A -85,B 0,C 180,E1 -6028.885,E2 -6028.885} C_VEL
LIN {X 0,Y 496.074,Z 484.524,A -85,B 0,C 180,E1 -6029.797,E2 -6029.797} C_VEL
LIN {X 0,Y 495.782,Z 492.345,A -85,B 0,C 180,E1 -6030.813,E2 -6030.813} C_VEL
LIN {X 0,Y 495.505,Z 500.027,A -85,B 0,C 180,E1 -6032.032,E2 -6032.032} C_VEL
LIN {X 0,Y 495.289,Z 506.191,A -85,B 0,C 180,E1 -6033.254,E2 -6033.254} C_VEL
LIN {X 0,Y 495.154,Z 511.106,A -85,B 0,C 180,E1 -6034.478,E2 -6034.478} C_VEL
LIN {X 0,Y 495.139,Z 514.91,A -85,B 0,C 180,E1 -6035.702,E2 -6035.702} C_VEL
LIN {X 0,Y 495.12,Z 516.876,A -85,B 0,C 180,E1 -6036.521,E2 -6036.521} C_VEL
LIN {X 0,Y 495.012,Z 518.441,A -85,B 0,C 180,E1 -6037.341,E2 -6037.341} C_VEL
LIN {X 0,Y 494.991,Z 519.568,A -85,B 0,C 180,E1 -6038.163,E2 -6038.163} C_VEL
LIN {X 0,Y 494.934,Z 520.594,A -85,B 0,C 180,E1 -6039.811,E2 -6039.811} C_VEL
LIN {X 0,Y 494.971,Z 520.525,A -85,B 0,C 180,E1 -6040.637,E2 -6040.637} C_VEL
LIN {X 0,Y 495.006,Z 519.913,A -85,B 0,C 180,E1 -6041.58,E2 -6041.58} C_VEL
LIN {X 0,Y 494.973,Z 517.778,A -85,B 0,C 180,E1 -6043.131,E2 -6043.131} C_VEL
LIN {X 0,Y 495.099,Z 514.942,A -85,B 0,C 180,E1 -6044.384,E2 -6044.384} C_VEL
LIN {X 0,Y 495.176,Z 511.023,A -85,B 0,C 180,E1 -6045.645,E2 -6045.645} C_VEL
LIN {X 0,Y 495.333,Z 505.898,A -85,B 0,C 180,E1 -6046.91,E2 -6046.91} C_VEL
LIN {X 0,Y 495.575,Z 499.367,A -85,B 0,C 180,E1 -6048.18,E2 -6048.18} C_VEL
LIN {X 0,Y 495.831,Z 491.099,A -85,B 0,C 180,E1 -6049.457,E2 -6049.457} C_VEL
LIN {X 0,Y 496.168,Z 482.589,A -85,B 0,C 180,E1 -6050.522,E2 -6050.522} C_VEL
LIN {X 0,Y 496.508,Z 473.332,A -85,B 0,C 180,E1 -6051.474,E2 -6051.474} C_VEL
LIN {X 0,Y 496.895,Z 462.91,A -85,B 0,C 180,E1 -6052.341,E2 -6052.341} C_VEL
LIN {X 0,Y 497.306,Z 451.571,A -85,B 0,C 180,E1 -6053.089,E2 -6053.089} C_VEL
LIN {X 0,Y 497.604,Z 438.86,A -85,B 0,C 180,E1 -6053.736,E2 -6053.736} C_VEL
LIN {X 0,Y 497.84,Z 426.122,A -85,B 0,C 180,E1 -6054.194,E2 -6054.194} C_VEL
LIN {X 0,Y 497.979,Z 414.714,A -85,B 0,C 180,E1 -6054.465,E2 -6054.465} C_VEL
LIN {X 0,Y 498.614,Z 322.184,A -85,B 0,C 180,E1 -6055.815,E2 -6055.815} C_VEL
LIN {X 0,Y 496.285,Z 309.808,A -85,B 0,C 180,E1 -6056.104,E2 -6056.104} C_VEL
LIN {X 0,Y 496.484,Z 294.376,A -85,B 0,C 180,E1 -6059.001,E2 -6059.001} C_VEL
LIN {X 0,Y 495.816,Z 288.729,A -85,B 0,C 180,E1 -6060.118,E2 -6060.118} C_VEL
LIN {X 0,Y 495.759,Z 288.73,A -85,B 0,C 180,E1 -6063.564,E2 -6063.564} C_VEL
LIN {X 0,Y 495.727,Z 288.734,A -85,B 0,C 180,E1 -6066.544,E2 -6066.544} C_VEL
LIN {X 0,Y 495.756,Z 288.728,A -85,B 0,C 180,E1 -6069.638,E2 -6069.638} C_VEL
LIN {X 0,Y 495.737,Z 288.736,A -85,B 0,C 180,E1 -6072.507,E2 -6072.507} C_VEL
LIN {X 0,Y 495.736,Z 288.732,A -85,B 0,C 180,E1 -6075.141,E2 -6075.141} C_VEL
LIN {X 0,Y 495.755,Z 288.729,A -85,B 0,C 180,E1 -6078.219,E2 -6078.219} C_VEL
LIN {X 0,Y 495.749,Z 288.727,A -85,B 0,C 180,E1 -6081.408,E2 -6081.408} C_VEL
LIN {X 0,Y 495.748,Z 288.728,A -85,B 0,C 180,E1 -6084.462,E2 -6084.462} C_VEL
LIN {X 0,Y 495.766,Z 288.726,A -85,B 0,C 180,E1 -6087.406,E2 -6087.406} C_VEL
LIN {X 0,Y 495.765,Z 288.722,A -85,B 0,C 180,E1 -6090.254,E2 -6090.254} C_VEL
LIN {X 0,Y 495.822,Z 288.722,A -85,B 0,C 180,E1 -6093.251,E2 -6093.251} C_VEL
LIN {X 0,Y 495.747,Z 288.726,A -85,B 0,C 180,E1 -6095.725,E2 -6095.725} C_VEL
LIN {X 0,Y 495.741,Z 288.727,A -85,B 0,C 180,E1 -6098.371,E2 -6098.371} C_VEL
LIN {X 0,Y 495.782,Z 288.722,A -85,B 0,C 180,E1 -6100.972,E2 -6100.972} C_VEL
LIN {X 0,Y 495.777,Z 288.731,A -85,B 0,C 180,E1 -6103.53,E2 -6103.53} C_VEL
LIN {X 0,Y 495.792,Z 288.725,A -85,B 0,C 180,E1 -6106.056,E2 -6106.056} C_VEL
LIN {X 0,Y 495.85,Z 288.712,A -85,B 0,C 180,E1 -6108.555,E2 -6108.555} C_VEL
LIN {X 0,Y 495.872,Z 288.719,A -85,B 0,C 180,E1 -6111.852,E2 -6111.852} C_VEL
LIN {X 0,Y 495.887,Z 288.712,A -85,B 0,C 180,E1 -6114.307,E2 -6114.307} C_VEL
LIN {X 0,Y 495.993,Z 288.699,A -85,B 0,C 180,E1 -6117.564,E2 -6117.564} C_VEL
LIN {X 0,Y 495.982,Z 288.698,A -85,B 0,C 180,E1 -6120.812,E2 -6120.812} C_VEL
LIN {X 0,Y 495.992,Z 288.698,A -85,B 0,C 180,E1 -6122.436,E2 -6122.436} C_VEL
LIN {X 0,Y 495.888,Z 288.711,A -85,B 0,C 180,E1 -6125.694,E2 -6125.694} C_VEL
LIN {X 0,Y 495.872,Z 288.715,A -85,B 0,C 180,E1 -6128.148,E2 -6128.148} C_VEL
LIN {X 0,Y 495.851,Z 288.711,A -85,B 0,C 180,E1 -6131.445,E2 -6131.445} C_VEL
LIN {X 0,Y 495.79,Z 288.724,A -85,B 0,C 180,E1 -6134.783,E2 -6134.783} C_VEL
LIN {X 0,Y 495.781,Z 288.723,A -85,B 0,C 180,E1 -6137.319,E2 -6137.319} C_VEL
LIN {X 0,Y 495.77,Z 288.723,A -85,B 0,C 180,E1 -6139.891,E2 -6139.891} C_VEL
LIN {X 0,Y 495.76,Z 288.732,A -85,B 0,C 180,E1 -6142.861,E2 -6142.861} C_VEL
LIN {X 0,Y 495.791,Z 288.722,A -85,B 0,C 180,E1 -6146.068,E2 -6146.068} C_VEL
LIN {X 0,Y 495.772,Z 288.73,A -85,B 0,C 180,E1 -6148.815,E2 -6148.815} C_VEL
LIN {X 0,Y 495.755,Z 288.726,A -85,B 0,C 180,E1 -6151.725,E2 -6151.725} C_VEL
LIN {X 0,Y 495.769,Z 288.728,A -85,B 0,C 180,E1 -6154.694,E2 -6154.694} C_VEL
LIN {X 0,Y 495.73,Z 288.733,A -85,B 0,C 180,E1 -6157.562,E2 -6157.562} C_VEL
LIN {X 0,Y 495.767,Z 288.719,A -85,B 0,C 180,E1 -6160.7,E2 -6160.7} C_VEL
LIN {X 0,Y 495.729,Z 288.73,A -85,B 0,C 180,E1 -6164.002,E2 -6164.002} C_VEL
LIN {X 0,Y 495.726,Z 288.734,A -85,B 0,C 180,E1 -6167.117,E2 -6167.117} C_VEL
LIN {X 0,Y 495.76,Z 288.73,A -85,B 0,C 180,E1 -6169.953,E2 -6169.953} C_VEL
LIN {X 0,Y 495.729,Z 288.728,A -85,B 0,C 180,E1 -6172.553,E2 -6172.553} C_VEL
LIN {X 0,Y 495.78,Z 288.729,A -85,B 0,C 180,E1 -6175.457,E2 -6175.457} C_VEL
LIN {X 0,Y 495.758,Z 288.73,A -85,B 0,C 180,E1 -6178.364,E2 -6178.364} C_VEL
LIN {X 0,Y 495.789,Z 288.728,A -85,B 0,C 180,E1 -6181.507,E2 -6181.507} C_VEL
LIN {X 0,Y 495.822,Z 288.724,A -85,B 0,C 180,E1 -6184.61,E2 -6184.61} C_VEL
LIN {X 0,Y 495.821,Z 288.83,A -85,B 0,C 180,E1 -6184.722,E2 -6184.722} C_VEL
LIN {X 0,Y 497.48,Z 297.393,A -85,B 0,C 180,E1 -6186.258,E2 -6186.258} C_VEL
LIN {X 0,Y 497.499,Z 305.264,A -85,B 0,C 180,E1 -6187.578,E2 -6187.578} C_VEL
LIN {X 0,Y 496.816,Z 324.93,A -85,B 0,C 180,E1 -6190.798,E2 -6190.798} C_VEL
LIN {X 0,Y 496.243,Z 344.506,A -85,B 0,C 180,E1 -6193.955,E2 -6193.955} C_VEL
LIN {X 0,Y 498.497,Z 360.565,A -85,B 0,C 180,E1 -6194.269,E2 -6194.269} C_VEL
LIN {X 0,Y 497.965,Z 452.79,A -85,B 0,C 180,E1 -6195.622,E2 -6195.622} C_VEL
LIN {X 0,Y 497.696,Z 465.357,A -85,B 0,C 180,E1 -6195.954,E2 -6195.954} C_VEL
LIN {X 0,Y 497.321,Z 478.319,A -85,B 0,C 180,E1 -6196.464,E2 -6196.464} C_VEL
LIN {X 0,Y 496.932,Z 490.579,A -85,B 0,C 180,E1 -6197.126,E2 -6197.126} C_VEL
LIN {X 0,Y 496.587,Z 502.259,A -85,B 0,C 180,E1 -6197.951,E2 -6197.951} C_VEL
LIN {X 0,Y 496.205,Z 512.733,A -85,B 0,C 180,E1 -6198.873,E2 -6198.873} C_VEL
LIN {X 0,Y 495.848,Z 521.297,A -85,B 0,C 180,E1 -6199.795,E2 -6199.795} C_VEL
LIN {X 0,Y 495.564,Z 529.202,A -85,B 0,C 180,E1 -6200.819,E2 -6200.819} C_VEL
LIN {X 0,Y 495.342,Z 536.926,A -85,B 0,C 180,E1 -6202.048,E2 -6202.048} C_VEL
LIN {X 0,Y 495.165,Z 544.046,A -85,B 0,C 180,E1 -6203.48,E2 -6203.48} C_VEL
LIN {X 0,Y 495.106,Z 548.786,A -85,B 0,C 180,E1 -6204.706,E2 -6204.706} C_VEL
LIN {X 0,Y 495.033,Z 552.406,A -85,B 0,C 180,E1 -6205.929,E2 -6205.929} C_VEL
LIN {X 0,Y 495.042,Z 554.276,A -85,B 0,C 180,E1 -6206.744,E2 -6206.744} C_VEL
LIN {X 0,Y 494.998,Z 555.677,A -85,B 0,C 180,E1 -6207.559,E2 -6207.559} C_VEL
LIN {X 0,Y 494.962,Z 556.676,A -85,B 0,C 180,E1 -6208.372,E2 -6208.372} C_VEL
LIN {X 0,Y 494.901,Z 557.505,A -85,B 0,C 180,E1 -6210,E2 -6210} C_VEL
LIN {X 0,Y 494.962,Z 556.686,A -85,B 0,C 180,E1 -6211.627,E2 -6211.627} C_VEL
LIN {X 0,Y 494.998,Z 555.692,A -85,B 0,C 180,E1 -6212.441,E2 -6212.441} C_VEL
LIN {X 0,Y 495.042,Z 554.296,A -85,B 0,C 180,E1 -6213.255,E2 -6213.255} C_VEL
LIN {X 0,Y 495.008,Z 551.353,A -85,B 0,C 180,E1 -6214.478,E2 -6214.478} C_VEL
LIN {X 0,Y 495.125,Z 547.375,A -85,B 0,C 180,E1 -6215.702,E2 -6215.702} C_VEL
LIN {X 0,Y 495.253,Z 541.253,A -85,B 0,C 180,E1 -6217.132,E2 -6217.132} C_VEL
LIN {X 0,Y 495.424,Z 534.562,A -85,B 0,C 180,E1 -6218.36,E2 -6218.36} C_VEL
LIN {X 0,Y 495.678,Z 526.263,A -85,B 0,C 180,E1 -6219.59,E2 -6219.59} C_VEL
LIN {X 0,Y 495.983,Z 517.756,A -85,B 0,C 180,E1 -6220.615,E2 -6220.615} C_VEL
LIN {X 0,Y 496.413,Z 507.248,A -85,B 0,C 180,E1 -6221.639,E2 -6221.639} C_VEL
LIN {X 0,Y 496.786,Z 495.725,A -85,B 0,C 180,E1 -6222.54,E2 -6222.54} C_VEL
LIN {X 0,Y 497.153,Z 483.52,A -85,B 0,C 180,E1 -6223.28,E2 -6223.28} C_VEL
LIN {X 0,Y 497.533,Z 471.138,A -85,B 0,C 180,E1 -6223.842,E2 -6223.842} C_VEL
LIN {X 0,Y 497.806,Z 458.414,A -85,B 0,C 180,E1 -6224.251,E2 -6224.251} C_VEL
LIN {X 0,Y 498.038,Z 445.054,A -85,B 0,C 180,E1 -6224.505,E2 -6224.505} C_VEL
LIN {X 0,Y 498.439,Z 358.963,A -85,B 0,C 180,E1 -6225.753,E2 -6225.753} C_VEL
LIN {X 0,Y 496.253,Z 344.621,A -85,B 0,C 180,E1 -6226.036,E2 -6226.036} C_VEL
LIN {X 0,Y 496.762,Z 326.281,A -85,B 0,C 180,E1 -6228.989,E2 -6228.989} C_VEL
LIN {X 0,Y 497.423,Z 306.52,A -85,B 0,C 180,E1 -6232.206,E2 -6232.206} C_VEL
LIN {X 0,Y 497.628,Z 298.716,A -85,B 0,C 180,E1 -6233.491,E2 -6233.491} C_VEL
LIN {X 0,Y 495.825,Z 288.725,A -85,B 0,C 180,E1 -6235.277,E2 -6235.277} C_VEL
LIN {X 0,Y 495.782,Z 288.731,A -85,B 0,C 180,E1 -6237.891,E2 -6237.891} C_VEL
LIN {X 0,Y 495.752,Z 288.728,A -85,B 0,C 180,E1 -6240.687,E2 -6240.687} C_VEL
LIN {X 0,Y 495.758,Z 288.727,A -85,B 0,C 180,E1 -6243.564,E2 -6243.564} C_VEL
LIN {X 0,Y 495.727,Z 288.734,A -85,B 0,C 180,E1 -6246.543,E2 -6246.543} C_VEL
LIN {X 0,Y 495.755,Z 288.727,A -85,B 0,C 180,E1 -6249.637,E2 -6249.637} C_VEL
LIN {X 0,Y 495.736,Z 288.737,A -85,B 0,C 180,E1 -6252.506,E2 -6252.506} C_VEL
LIN {X 0,Y 495.735,Z 288.73,A -85,B 0,C 180,E1 -6255.14,E2 -6255.14} C_VEL
LIN {X 0,Y 495.754,Z 288.73,A -85,B 0,C 180,E1 -6258.218,E2 -6258.218} C_VEL
LIN {X 0,Y 495.747,Z 288.727,A -85,B 0,C 180,E1 -6261.408,E2 -6261.408} C_VEL
LIN {X 0,Y 495.745,Z 288.732,A -85,B 0,C 180,E1 -6264.462,E2 -6264.462} C_VEL
LIN {X 0,Y 495.764,Z 288.727,A -85,B 0,C 180,E1 -6267.405,E2 -6267.405} C_VEL
LIN {X 0,Y 495.762,Z 288.726,A -85,B 0,C 180,E1 -6270.253,E2 -6270.253} C_VEL
LIN {X 0,Y 495.819,Z 288.723,A -85,B 0,C 180,E1 -6273.25,E2 -6273.25} C_VEL
LIN {X 0,Y 495.748,Z 288.728,A -85,B 0,C 180,E1 -6275.725,E2 -6275.725} C_VEL
LIN {X 0,Y 495.738,Z 288.728,A -85,B 0,C 180,E1 -6278.371,E2 -6278.371} C_VEL
LIN {X 0,Y 495.78,Z 288.729,A -85,B 0,C 180,E1 -6280.971,E2 -6280.971} C_VEL
LIN {X 0,Y 495.774,Z 288.729,A -85,B 0,C 180,E1 -6283.53,E2 -6283.53} C_VEL
LIN {X 0,Y 495.793,Z 288.722,A -85,B 0,C 180,E1 -6286.055,E2 -6286.055} C_VEL
LIN {X 0,Y 495.846,Z 288.715,A -85,B 0,C 180,E1 -6288.555,E2 -6288.555} C_VEL
LIN {X 0,Y 495.868,Z 288.716,A -85,B 0,C 180,E1 -6291.852,E2 -6291.852} C_VEL
LIN {X 0,Y 495.887,Z 288.71,A -85,B 0,C 180,E1 -6294.306,E2 -6294.306} C_VEL
LIN {X 0,Y 495.986,Z 288.705,A -85,B 0,C 180,E1 -6297.563,E2 -6297.563} C_VEL
LIN {X 0,Y 495.991,Z 288.702,A -85,B 0,C 180,E1 -6300,E2 -6300} C_VEL
LIN {X 0,Y 495.987,Z 288.698,A -85,B 0,C 180,E1 -6302.436,E2 -6302.436} C_VEL
LIN {X 0,Y 495.877,Z 288.717,A -85,B 0,C 180,E1 -6305.694,E2 -6305.694} C_VEL
LIN {X 0,Y 495.836,Z 288.716,A -85,B 0,C 180,E1 -6308.97,E2 -6308.97} C_VEL
LIN {X 0,Y 495.822,Z 288.727,A -85,B 0,C 180,E1 -6312.035,E2 -6312.035} C_VEL
LIN {X 0,Y 495.818,Z 288.719,A -85,B 0,C 180,E1 -6315.452,E2 -6315.452} C_VEL
LIN {X 0,Y 495.773,Z 288.733,A -85,B 0,C 180,E1 -6318.237,E2 -6318.237} C_VEL
LIN {X 0,Y 495.768,Z 288.727,A -85,B 0,C 180,E1 -6320.756,E2 -6320.756} C_VEL
LIN {X 0,Y 495.737,Z 288.728,A -85,B 0,C 180,E1 -6323.388,E2 -6323.388} C_VEL
LIN {X 0,Y 495.806,Z 288.724,A -85,B 0,C 180,E1 -6326.747,E2 -6326.747} C_VEL
LIN {X 0,Y 495.76,Z 288.726,A -85,B 0,C 180,E1 -6329.747,E2 -6329.747} C_VEL
LIN {X 0,Y 495.762,Z 288.734,A -85,B 0,C 180,E1 -6332.595,E2 -6332.595} C_VEL
LIN {X 0,Y 495.742,Z 288.728,A -85,B 0,C 180,E1 -6335.538,E2 -6335.538} C_VEL
LIN {X 0,Y 495.755,Z 288.735,A -85,B 0,C 180,E1 -6338.768,E2 -6338.768} C_VEL
LIN {X 0,Y 495.751,Z 288.726,A -85,B 0,C 180,E1 -6341.782,E2 -6341.782} C_VEL
LIN {X 0,Y 495.745,Z 288.734,A -85,B 0,C 180,E1 -6345.14,E2 -6345.14} C_VEL
LIN {X 0,Y 495.739,Z 288.728,A -85,B 0,C 180,E1 -6348.218,E2 -6348.218} C_VEL
LIN {X 0,Y 495.742,Z 288.733,A -85,B 0,C 180,E1 -6351.408,E2 -6351.408} C_VEL
LIN {X 0,Y 495.743,Z 288.728,A -85,B 0,C 180,E1 -6354.463,E2 -6354.463} C_VEL
LIN {X 0,Y 495.762,Z 288.733,A -85,B 0,C 180,E1 -6357.406,E2 -6357.406} C_VEL
LIN {X 0,Y 495.756,Z 288.726,A -85,B 0,C 180,E1 -6360.254,E2 -6360.254} C_VEL
LIN {X 0,Y 495.726,Z 288.731,A -85,B 0,C 180,E1 -6360.738,E2 -6360.738} C_VEL
LIN {X 0,Y 495.048,Z 288.823,A -85,B 0,C 180,E1 -6361.417,E2 -6361.417} C_VEL
LIN {X 0,Y 492.171,Z 289.178,A -85,B 0,C 180,E1 -6362.519,E2 -6362.519} C_VEL
LIN {X 0,Y 489.753,Z 289.482,A -85,B 0,C 180,E1 -6363.407,E2 -6363.407} C_VEL
LIN {X 0,Y 488.73,Z 289.603,A -85,B 0,C 180,E1 -6364.093,E2 -6364.093} C_VEL
LIN {X 0,Y 488.654,Z 289.611,A -85,B 0,C 180,E1 -6364.325,E2 -6364.325} C_VEL
LIN {X 0,Y 488.719,Z 289.606,A -85,B 0,C 180,E1 -6367.154,E2 -6367.154} C_VEL
LIN {X 0,Y 488.722,Z 289.609,A -85,B 0,C 180,E1 -6369.811,E2 -6369.811} C_VEL
LIN {X 0,Y 488.699,Z 289.606,A -85,B 0,C 180,E1 -6372.423,E2 -6372.423} C_VEL
LIN {X 0,Y 488.759,Z 289.598,A -85,B 0,C 180,E1 -6375,E2 -6375} C_VEL
LIN {X 0,Y 488.782,Z 289.602,A -85,B 0,C 180,E1 -6378.387,E2 -6378.387} C_VEL
LIN {X 0,Y 488.748,Z 289.765,A -85,B 0,C 180,E1 -6379.802,E2 -6379.802} C_VEL
LIN {X 0,Y 489.507,Z 295.272,A -85,B 0,C 180,E1 -6380.914,E2 -6380.914} C_VEL
LIN {X 0,Y 489.333,Z 308.111,A -85,B 0,C 180,E1 -6383.403,E2 -6383.403} C_VEL
LIN {X 0,Y 489.24,Z 310.145,A -85,B 0,C 180,E1 -6383.79,E2 -6383.79} C_VEL
LIN {X 0,Y 491.755,Z 323.135,A -85,B 0,C 180,E1 -6384.079,E2 -6384.079} C_VEL
LIN {X 0,Y 491.114,Z 417.685,A -85,B 0,C 180,E1 -6385.486,E2 -6385.486} C_VEL
LIN {X 0,Y 490.877,Z 430.631,A -85,B 0,C 180,E1 -6385.844,E2 -6385.844} C_VEL
LIN {X 0,Y 490.646,Z 443.096,A -85,B 0,C 180,E1 -6386.356,E2 -6386.356} C_VEL
LIN {X 0,Y 490.266,Z 455.056,A -85,B 0,C 180,E1 -6387.022,E2 -6387.022} C_VEL
LIN {X 0,Y 489.766,Z 466.456,A -85,B 0,C 180,E1 -6387.842,E2 -6387.842} C_VEL
LIN {X 0,Y 489.329,Z 476.723,A -85,B 0,C 180,E1 -6388.766,E2 -6388.766} C_VEL
LIN {X 0,Y 489.036,Z 485.97,A -85,B 0,C 180,E1 -6389.794,E2 -6389.794} C_VEL
LIN {X 0,Y 488.672,Z 494.926,A -85,B 0,C 180,E1 -6391.03,E2 -6391.03} C_VEL
LIN {X 0,Y 488.366,Z 502.164,A -85,B 0,C 180,E1 -6392.268,E2 -6392.268} C_VEL
LIN {X 0,Y 488.199,Z 508.81,A -85,B 0,C 180,E1 -6393.715,E2 -6393.715} C_VEL
LIN {X 0,Y 488.002,Z 513.222,A -85,B 0,C 180,E1 -6394.957,E2 -6394.957} C_VEL
LIN {X 0,Y 488.048,Z 517.156,A -85,B 0,C 180,E1 -6396.479,E2 -6396.479} C_VEL
LIN {X 0,Y 487.924,Z 518.936,A -85,B 0,C 180,E1 -6397.449,E2 -6397.449} C_VEL
LIN {X 0,Y 487.908,Z 519.972,A -85,B 0,C 180,E1 -6398.282,E2 -6398.282} C_VEL
LIN {X 0,Y 487.866,Z 520.886,A -85,B 0,C 180,E1 -6399.955,E2 -6399.955} C_VEL
LIN {X 0,Y 487.882,Z 520.73,A -85,B 0,C 180,E1 -6400.793,E2 -6400.793} C_VEL
LIN {X 0,Y 487.927,Z 520.148,A -85,B 0,C 180,E1 -6401.634,E2 -6401.634} C_VEL
LIN {X 0,Y 487.866,Z 519.17,A -85,B 0,C 180,E1 -6402.479,E2 -6402.479} C_VEL
LIN {X 0,Y 487.904,Z 517.783,A -85,B 0,C 180,E1 -6403.325,E2 -6403.325} C_VEL
LIN {X 0,Y 488.028,Z 514.828,A -85,B 0,C 180,E1 -6404.597,E2 -6404.597} C_VEL
LIN {X 0,Y 488.137,Z 510.776,A -85,B 0,C 180,E1 -6405.876,E2 -6405.876} C_VEL
LIN {X 0,Y 488.362,Z 504.449,A -85,B 0,C 180,E1 -6407.374,E2 -6407.374} C_VEL
LIN {X 0,Y 488.587,Z 497.482,A -85,B 0,C 180,E1 -6408.666,E2 -6408.666} C_VEL
LIN {X 0,Y 488.866,Z 490.307,A -85,B 0,C 180,E1 -6409.745,E2 -6409.745} C_VEL
LIN {X 0,Y 489.275,Z 481.109,A -85,B 0,C 180,E1 -6410.876,E2 -6410.876} C_VEL
LIN {X 0,Y 489.676,Z 470.634,A -85,B 0,C 180,E1 -6411.911,E2 -6411.911} C_VEL
LIN {X 0,Y 490.119,Z 459.686,A -85,B 0,C 180,E1 -6412.778,E2 -6412.778} C_VEL
LIN {X 0,Y 490.523,Z 447.78,A -85,B 0,C 180,E1 -6413.514,E2 -6413.514} C_VEL
LIN {X 0,Y 490.763,Z 435.532,A -85,B 0,C 180,E1 -6414.088,E2 -6414.088} C_VEL
LIN {X 0,Y 490.946,Z 423.134,A -85,B 0,C 180,E1 -6414.5,E2 -6414.5} C_VEL
LIN {X 0,Y 491.171,Z 409.398,A -85,B 0,C 180,E1 -6414.77,E2 -6414.77} C_VEL
LIN {X 0,Y 491.775,Z 322.868,A -85,B 0,C 180,E1 -6416.044,E2 -6416.044} C_VEL
LIN {X 0,Y 489.31,Z 310.113,A -85,B 0,C 180,E1 -6416.335,E2 -6416.335} C_VEL
LIN {X 0,Y 489.532,Z 294.925,A -85,B 0,C 180,E1 -6419.217,E2 -6419.217} C_VEL
LIN {X 0,Y 488.751,Z 289.608,A -85,B 0,C 180,E1 -6420.295,E2 -6420.295} C_VEL
LIN {X 0,Y 488.734,Z 289.605,A -85,B 0,C 180,E1 -6423.484,E2 -6423.484} C_VEL
LIN {X 0,Y 488.682,Z 289.615,A -85,B 0,C 180,E1 -6426.355,E2 -6426.355} C_VEL
LIN {X 0,Y 488.7,Z 289.608,A -85,B 0,C 180,E1 -6429.254,E2 -6429.254} C_VEL
LIN {X 0,Y 488.706,Z 289.606,A -85,B 0,C 180,E1 -6431.6,E2 -6431.6} C_VEL
LIN {X 0,Y 488.7,Z 289.613,A -85,B 0,C 180,E1 -6434.803,E2 -6434.803} C_VEL
LIN {X 0,Y 488.691,Z 289.607,A -85,B 0,C 180,E1 -6437.475,E2 -6437.475} C_VEL
LIN {X 0,Y 488.732,Z 289.601,A -85,B 0,C 180,E1 -6439.677,E2 -6439.677} C_VEL
LIN {X 0,Y 488.678,Z 289.615,A -85,B 0,C 180,E1 -6442.841,E2 -6442.841} C_VEL
LIN {X 0,Y 488.73,Z 289.6,A -85,B 0,C 180,E1 -6445.887,E2 -6445.887} C_VEL
LIN {X 0,Y 488.691,Z 289.609,A -85,B 0,C 180,E1 -6448.82,E2 -6448.82} C_VEL
LIN {X 0,Y 488.743,Z 289.598,A -85,B 0,C 180,E1 -6451.671,E2 -6451.671} C_VEL
LIN {X 0,Y 488.739,Z 289.599,A -85,B 0,C 180,E1 -6454.444,E2 -6454.444} C_VEL
LIN {X 0,Y 488.722,Z 289.604,A -85,B 0,C 180,E1 -6457.153,E2 -6457.153} C_VEL
LIN {X 0,Y 488.724,Z 289.602,A -85,B 0,C 180,E1 -6459.811,E2 -6459.811} C_VEL
LIN {X 0,Y 488.728,Z 289.602,A -85,B 0,C 180,E1 -6462.423,E2 -6462.423} C_VEL
LIN {X 0,Y 488.761,Z 289.596,A -85,B 0,C 180,E1 -6465,E2 -6465} C_VEL
LIN {X 0,Y 488.804,Z 289.591,A -85,B 0,C 180,E1 -6468.388,E2 -6468.388} C_VEL
LIN {X 0,Y 488.817,Z 289.599,A -85,B 0,C 180,E1 -6471.734,E2 -6471.734} C_VEL
LIN {X 0,Y 488.846,Z 289.59,A -85,B 0,C 180,E1 -6474.224,E2 -6474.224} C_VEL
LIN {X 0,Y 488.96,Z 289.575,A -85,B 0,C 180,E1 -6477.529,E2 -6477.529} C_VEL
LIN {X 0,Y 488.933,Z 289.576,A -85,B 0,C 180,E1 -6480.824,E2 -6480.824} C_VEL
LIN {X 0,Y 488.96,Z 289.574,A -85,B 0,C 180,E1 -6482.472,E2 -6482.472} C_VEL
LIN {X 0,Y 488.846,Z 289.589,A -85,B 0,C 180,E1 -6485.776,E2 -6485.776} C_VEL
LIN {X 0,Y 488.817,Z 289.595,A -85,B 0,C 180,E1 -6488.267,E2 -6488.267} C_VEL
LIN {X 0,Y 488.805,Z 289.589,A -85,B 0,C 180,E1 -6491.613,E2 -6491.613} C_VEL
LIN {X 0,Y 488.762,Z 289.597,A -85,B 0,C 180,E1 -6495.001,E2 -6495.001} C_VEL
LIN {X 0,Y 488.755,Z 289.604,A -85,B 0,C 180,E1 -6498.442,E2 -6498.442} C_VEL
LIN {X 0,Y 488.707,Z 289.607,A -85,B 0,C 180,E1 -6501.071,E2 -6501.071} C_VEL
LIN {X 0,Y 488.689,Z 289.605,A -85,B 0,C 180,E1 -6503.746,E2 -6503.746} C_VEL
LIN {X 0,Y 488.792,Z 289.601,A -85,B 0,C 180,E1 -6506.944,E2 -6506.944} C_VEL
LIN {X 0,Y 488.71,Z 289.606,A -85,B 0,C 180,E1 -6510.363,E2 -6510.363} C_VEL
LIN {X 0,Y 488.735,Z 289.604,A -85,B 0,C 180,E1 -6513.484,E2 -6513.484} C_VEL
LIN {X 0,Y 488.683,Z 289.605,A -85,B 0,C 180,E1 -6516.355,E2 -6516.355} C_VEL
LIN {X 0,Y 488.702,Z 289.606,A -85,B 0,C 180,E1 -6519.254,E2 -6519.254} C_VEL
LIN {X 0,Y 488.708,Z 289.609,A -85,B 0,C 180,E1 -6521.6,E2 -6521.6} C_VEL
LIN {X 0,Y 488.702,Z 289.605,A -85,B 0,C 180,E1 -6524.803,E2 -6524.803} C_VEL
LIN {X 0,Y 488.693,Z 289.614,A -85,B 0,C 180,E1 -6527.475,E2 -6527.475} C_VEL
LIN {X 0,Y 488.735,Z 289.609,A -85,B 0,C 180,E1 -6529.677,E2 -6529.677} C_VEL
LIN {X 0,Y 488.681,Z 289.606,A -85,B 0,C 180,E1 -6532.841,E2 -6532.841} C_VEL
LIN {X 0,Y 488.732,Z 289.609,A -85,B 0,C 180,E1 -6535.887,E2 -6535.887} C_VEL
LIN {X 0,Y 488.694,Z 289.608,A -85,B 0,C 180,E1 -6538.82,E2 -6538.82} C_VEL
LIN {X 0,Y 488.746,Z 289.606,A -85,B 0,C 180,E1 -6541.671,E2 -6541.671} C_VEL
LIN {X 0,Y 488.813,Z 289.728,A -85,B 0,C 180,E1 -6544.512,E2 -6544.512} C_VEL
LIN {X 0,Y 490.656,Z 299.867,A -85,B 0,C 180,E1 -6546.355,E2 -6546.355} C_VEL
LIN {X 0,Y 490.385,Z 310.341,A -85,B 0,C 180,E1 -6548.123,E2 -6548.123} C_VEL
LIN {X 0,Y 489.736,Z 329.429,A -85,B 0,C 180,E1 -6551.288,E2 -6551.288} C_VEL
LIN {X 0,Y 489.258,Z 344.235,A -85,B 0,C 180,E1 -6553.71,E2 -6553.71} C_VEL
LIN {X 0,Y 491.681,Z 360.857,A -85,B 0,C 180,E1 -6554.045,E2 -6554.045} C_VEL
LIN {X 0,Y 491.115,Z 452.758,A -85,B 0,C 180,E1 -6555.417,E2 -6555.417} C_VEL
LIN {X 0,Y 490.801,Z 465.994,A -85,B 0,C 180,E1 -6555.779,E2 -6555.779} C_VEL
LIN {X 0,Y 490.435,Z 478.145,A -85,B 0,C 180,E1 -6556.27,E2 -6556.27} C_VEL
LIN {X 0,Y 489.975,Z 490.673,A -85,B 0,C 180,E1 -6556.96,E2 -6556.96} C_VEL
LIN {X 0,Y 489.584,Z 502.023,A -85,B 0,C 180,E1 -6557.776,E2 -6557.776} C_VEL
LIN {X 0,Y 489.173,Z 512.478,A -85,B 0,C 180,E1 -6558.711,E2 -6558.711} C_VEL
LIN {X 0,Y 488.836,Z 521.036,A -85,B 0,C 180,E1 -6559.647,E2 -6559.647} C_VEL
LIN {X 0,Y 488.521,Z 528.937,A -85,B 0,C 180,E1 -6560.686,E2 -6560.686} C_VEL
LIN {X 0,Y 488.276,Z 536.658,A -85,B 0,C 180,E1 -6561.932,E2 -6561.932} C_VEL
LIN {X 0,Y 488.074,Z 543.776,A -85,B 0,C 180,E1 -6563.385,E2 -6563.385} C_VEL
LIN {X 0,Y 488.018,Z 548.517,A -85,B 0,C 180,E1 -6564.629,E2 -6564.629} C_VEL
LIN {X 0,Y 487.929,Z 552.139,A -85,B 0,C 180,E1 -6565.87,E2 -6565.87} C_VEL
LIN {X 0,Y 487.965,Z 554.01,A -85,B 0,C 180,E1 -6566.697,E2 -6566.697} C_VEL
LIN {X 0,Y 487.89,Z 556.412,A -85,B 0,C 180,E1 -6568.349,E2 -6568.349} C_VEL
LIN {X 0,Y 487.822,Z 557.242,A -85,B 0,C 180,E1 -6570,E2 -6570} C_VEL
LIN {X 0,Y 487.89,Z 556.423,A -85,B 0,C 180,E1 -6571.651,E2 -6571.651} C_VEL
LIN {X 0,Y 487.964,Z 554.032,A -85,B 0,C 180,E1 -6573.302,E2 -6573.302} C_VEL
LIN {X 0,Y 487.92,Z 551.089,A -85,B 0,C 180,E1 -6574.544,E2 -6574.544} C_VEL
LIN {X 0,Y 488.021,Z 547.11,A -85,B 0,C 180,E1 -6575.785,E2 -6575.785} C_VEL
LIN {X 0,Y 488.18,Z 540.987,A -85,B 0,C 180,E1 -6577.236,E2 -6577.236} C_VEL
LIN {X 0,Y 488.357,Z 534.293,A -85,B 0,C 180,E1 -6578.482,E2 -6578.482} C_VEL
LIN {X 0,Y 488.647,Z 525.99,A -85,B 0,C 180,E1 -6579.729,E2 -6579.729} C_VEL
LIN {X 0,Y 488.992,Z 517.477,A -85,B 0,C 180,E1 -6580.768,E2 -6580.768} C_VEL
LIN {X 0,Y 489.428,Z 506.959,A -85,B 0,C 180,E1 -6581.807,E2 -6581.807} C_VEL
LIN {X 0,Y 489.811,Z 495.586,A -85,B 0,C 180,E1 -6582.71,E2 -6582.71} C_VEL
LIN {X 0,Y 490.237,Z 483.182,A -85,B 0,C 180,E1 -6583.471,E2 -6583.471} C_VEL
LIN {X 0,Y 490.642,Z 470.765,A -85,B 0,C 180,E1 -6584.04,E2 -6584.04} C_VEL
LIN {X 0,Y 490.936,Z 457.972,A -85,B 0,C 180,E1 -6584.455,E2 -6584.455} C_VEL
LIN {X 0,Y 491.152,Z 444.441,A -85,B 0,C 180,E1 -6584.713,E2 -6584.713} C_VEL
LIN {X 0,Y 491.579,Z 359.66,A -85,B 0,C 180,E1 -6585.958,E2 -6585.958} C_VEL
LIN {X 0,Y 489.259,Z 344.332,A -85,B 0,C 180,E1 -6586.267,E2 -6586.267} C_VEL
LIN {X 0,Y 489.801,Z 325.946,A -85,B 0,C 180,E1 -6589.269,E2 -6589.269} C_VEL
LIN {X 0,Y 490.473,Z 307.475,A -85,B 0,C 180,E1 -6592.316,E2 -6592.316} C_VEL
LIN {X 0,Y 490.619,Z 299.524,A -85,B 0,C 180,E1 -6593.646,E2 -6593.646} C_VEL
LIN {X 0,Y 488.794,Z 289.601,A -85,B 0,C 180,E1 -6595.42,E2 -6595.42} C_VEL
LIN {X 0,Y 488.745,Z 289.607,A -85,B 0,C 180,E1 -6598.328,E2 -6598.328} C_VEL
LIN {X 0,Y 488.692,Z 289.606,A -85,B 0,C 180,E1 -6601.179,E2 -6601.179} C_VEL
LIN {X 0,Y 488.73,Z 289.609,A -85,B 0,C 180,E1 -6604.112,E2 -6604.112} C_VEL
LIN {X 0,Y 488.678,Z 289.608,A -85,B 0,C 180,E1 -6607.158,E2 -6607.158} C_VEL
LIN {X 0,Y 488.717,Z 289.612,A -85,B 0,C 180,E1 -6610.344,E2 -6610.344} C_VEL
LIN {X 0,Y 488.682,Z 289.607,A -85,B 0,C 180,E1 -6613.654,E2 -6613.654} C_VEL
LIN {X 0,Y 488.682,Z 289.613,A -85,B 0,C 180,E1 -6616.345,E2 -6616.345} C_VEL
LIN {X 0,Y 488.73,Z 289.601,A -85,B 0,C 180,E1 -6619.676,E2 -6619.676} C_VEL
LIN {X 0,Y 488.676,Z 289.615,A -85,B 0,C 180,E1 -6622.841,E2 -6622.841} C_VEL
LIN {X 0,Y 488.727,Z 289.601,A -85,B 0,C 180,E1 -6625.887,E2 -6625.887} C_VEL
LIN {X 0,Y 488.689,Z 289.615,A -85,B 0,C 180,E1 -6628.82,E2 -6628.82} C_VEL
LIN {X 0,Y 488.741,Z 289.6,A -85,B 0,C 180,E1 -6631.671,E2 -6631.671} C_VEL
LIN {X 0,Y 488.744,Z 289.601,A -85,B 0,C 180,E1 -6634.444,E2 -6634.444} C_VEL
LIN {X 0,Y 488.72,Z 289.611,A -85,B 0,C 180,E1 -6637.153,E2 -6637.153} C_VEL
LIN {X 0,Y 488.72,Z 289.603,A -85,B 0,C 180,E1 -6639.81,E2 -6639.81} C_VEL
LIN {X 0,Y 488.729,Z 289.601,A -85,B 0,C 180,E1 -6642.423,E2 -6642.423} C_VEL
LIN {X 0,Y 488.76,Z 289.602,A -85,B 0,C 180,E1 -6644.999,E2 -6644.999} C_VEL
LIN {X 0,Y 488.8,Z 289.592,A -85,B 0,C 180,E1 -6648.387,E2 -6648.387} C_VEL
LIN {X 0,Y 488.813,Z 289.596,A -85,B 0,C 180,E1 -6651.733,E2 -6651.733} C_VEL
LIN {X 0,Y 488.847,Z 289.588,A -85,B 0,C 180,E1 -6654.224,E2 -6654.224} C_VEL
LIN {X 0,Y 488.954,Z 289.58,A -85,B 0,C 180,E1 -6657.528,E2 -6657.528} C_VEL
LIN {X 0,Y 488.963,Z 289.577,A -85,B 0,C 180,E1 -6660,E2 -6660} C_VEL
LIN {X 0,Y 488.955,Z 289.574,A -85,B 0,C 180,E1 -6662.471,E2 -6662.471} C_VEL
LIN {X 0,Y 488.834,Z 289.596,A -85,B 0,C 180,E1 -6665.776,E2 -6665.776} C_VEL
LIN {X 0,Y 488.811,Z 289.595,A -85,B 0,C 180,E1 -6668.266,E2 -6668.266} C_VEL
LIN {X 0,Y 488.8,Z 289.595,A -85,B 0,C 180,E1 -6671.612,E2 -6671.612} C_VEL
LIN {X 0,Y 488.755,Z 289.598,A -85,B 0,C 180,E1 -6675,E2 -6675} C_VEL
LIN {X 0,Y 488.741,Z 289.606,A -85,B 0,C 180,E1 -6678.443,E2 -6678.443} C_VEL
LIN {X 0,Y 488.701,Z 289.605,A -85,B 0,C 180,E1 -6681.071,E2 -6681.071} C_VEL
LIN {X 0,Y 488.674,Z 289.609,A -85,B 0,C 180,E1 -6683.746,E2 -6683.746} C_VEL
LIN {X 0,Y 488.745,Z 289.602,A -85,B 0,C 180,E1 -6686.934,E2 -6686.934} C_VEL
LIN {X 0,Y 488.718,Z 289.607,A -85,B 0,C 180,E1 -6690.22,E2 -6690.22} C_VEL
LIN {X 0,Y 488.729,Z 289.601,A -85,B 0,C 180,E1 -6693.484,E2 -6693.484} C_VEL
LIN {X 0,Y 488.677,Z 289.612,A -85,B 0,C 180,E1 -6696.355,E2 -6696.355} C_VEL
LIN {X 0,Y 488.692,Z 289.608,A -85,B 0,C 180,E1 -6699.255,E2 -6699.255} C_VEL
LIN {X 0,Y 488.702,Z 289.605,A -85,B 0,C 180,E1 -6701.6,E2 -6701.6} C_VEL
LIN {X 0,Y 488.708,Z 289.611,A -85,B 0,C 180,E1 -6704.802,E2 -6704.802} C_VEL
LIN {X 0,Y 488.663,Z 289.612,A -85,B 0,C 180,E1 -6707.472,E2 -6707.472} C_VEL
LIN {X 0,Y 488.689,Z 289.61,A -85,B 0,C 180,E1 -6710.745,E2 -6710.745} C_VEL
LIN {X 0,Y 488.673,Z 289.609,A -85,B 0,C 180,E1 -6713.868,E2 -6713.868} C_VEL
LIN {X 0,Y 488.732,Z 289.604,A -85,B 0,C 180,E1 -6716.877,E2 -6716.877} C_VEL
LIN {X 0,Y 488.716,Z 289.606,A -85,B 0,C 180,E1 -6719.781,E2 -6719.781} C_VEL
LIN {X 0,Y 488.695,Z 289.609,A -85,B 0,C 180,E1 -6723.079,E2 -6723.079} C_VEL
LIN {X 0,Y 488.654,Z 289.611,A -85,B 0,C 180,E1 -6724.325,E2 -6724.325} C_VEL
LIN {X 0,Y 488.012,Z 289.694,A -85,B 0,C 180,E1 -6725.013,E2 -6725.013} C_VEL
LIN {X 0,Y 485.179,Z 290.05,A -85,B 0,C 180,E1 -6726.131,E2 -6726.131} C_VEL
LIN {X 0,Y 482.765,Z 290.353,A -85,B 0,C 180,E1 -6727.032,E2 -6727.032} C_VEL
LIN {X 0,Y 481.722,Z 290.481,A -85,B 0,C 180,E1 -6727.728,E2 -6727.728} C_VEL
LIN {X 0,Y 481.634,Z 290.489,A -85,B 0,C 180,E1 -6727.963,E2 -6727.963} C_VEL
LIN {X 0,Y 481.699,Z 290.478,A -85,B 0,C 180,E1 -6730.393,E2 -6730.393} C_VEL
LIN {X 0,Y 481.665,Z 290.482,A -85,B 0,C 180,E1 -6733.033,E2 -6733.033} C_VEL
LIN {X 0,Y 481.684,Z 290.486,A -85,B 0,C 180,E1 -6735.639,E2 -6735.639} C_VEL
LIN {X 0,Y 481.733,Z 290.481,A -85,B 0,C 180,E1 -6738.215,E2 -6738.215} C_VEL
LIN {X 0,Y 481.689,Z 290.566,A -85,B 0,C 180,E1 -6739.651,E2 -6739.651} C_VEL
LIN {X 0,Y 482.518,Z 296.093,A -85,B 0,C 180,E1 -6740.781,E2 -6740.781} C_VEL
LIN {X 0,Y 482.374,Z 306.864,A -85,B 0,C 180,E1 -6742.887,E2 -6742.887} C_VEL
LIN {X 0,Y 482.297,Z 310.39,A -85,B 0,C 180,E1 -6743.568,E2 -6743.568} C_VEL
LIN {X 0,Y 484.957,Z 324.467,A -85,B 0,C 180,E1 -6743.878,E2 -6743.878} C_VEL
LIN {X 0,Y 484.22,Z 418.168,A -85,B 0,C 180,E1 -6745.291,E2 -6745.291} C_VEL
LIN {X 0,Y 483.965,Z 431.795,A -85,B 0,C 180,E1 -6745.68,E2 -6745.68} C_VEL
LIN {X 0,Y 483.719,Z 444.026,A -85,B 0,C 180,E1 -6746.199,E2 -6746.199} C_VEL
LIN {X 0,Y 483.336,Z 455.794,A -85,B 0,C 180,E1 -6746.875,E2 -6746.875} C_VEL
LIN {X 0,Y 482.8,Z 467.118,A -85,B 0,C 180,E1 -6747.706,E2 -6747.706} C_VEL
LIN {X 0,Y 482.335,Z 477.325,A -85,B 0,C 180,E1 -6748.644,E2 -6748.644} C_VEL
LIN {X 0,Y 482.041,Z 485.667,A -85,B 0,C 180,E1 -6749.583,E2 -6749.583} C_VEL
LIN {X 0,Y 481.671,Z 494.742,A -85,B 0,C 180,E1 -6750.836,E2 -6750.836} C_VEL
LIN {X 0,Y 481.341,Z 502.065,A -85,B 0,C 180,E1 -6752.092,E2 -6752.092} C_VEL
LIN {X 0,Y 481.171,Z 507.943,A -85,B 0,C 180,E1 -6753.35,E2 -6753.35} C_VEL
LIN {X 0,Y 480.968,Z 512.608,A -85,B 0,C 180,E1 -6754.61,E2 -6754.61} C_VEL
LIN {X 0,Y 480.973,Z 516.168,A -85,B 0,C 180,E1 -6755.871,E2 -6755.871} C_VEL
LIN {X 0,Y 480.941,Z 518.008,A -85,B 0,C 180,E1 -6756.714,E2 -6756.714} C_VEL
LIN {X 0,Y 480.805,Z 520.374,A -85,B 0,C 180,E1 -6758.405,E2 -6758.405} C_VEL
LIN {X 0,Y 480.749,Z 520.971,A -85,B 0,C 180,E1 -6759.254,E2 -6759.254} C_VEL
LIN {X 0,Y 480.772,Z 521.158,A -85,B 0,C 180,E1 -6760.103,E2 -6760.103} C_VEL
LIN {X 0,Y 480.84,Z 520.39,A -85,B 0,C 180,E1 -6761.685,E2 -6761.685} C_VEL
LIN {X 0,Y 480.788,Z 519.241,A -85,B 0,C 180,E1 -6762.666,E2 -6762.666} C_VEL
LIN {X 0,Y 480.826,Z 517.753,A -85,B 0,C 180,E1 -6763.525,E2 -6763.525} C_VEL
LIN {X 0,Y 480.975,Z 514.682,A -85,B 0,C 180,E1 -6764.816,E2 -6764.816} C_VEL
LIN {X 0,Y 481.087,Z 510.493,A -85,B 0,C 180,E1 -6766.115,E2 -6766.115} C_VEL
LIN {X 0,Y 481.355,Z 504.02,A -85,B 0,C 180,E1 -6767.636,E2 -6767.636} C_VEL
LIN {X 0,Y 481.647,Z 496.891,A -85,B 0,C 180,E1 -6768.945,E2 -6768.945} C_VEL
LIN {X 0,Y 481.971,Z 487.835,A -85,B 0,C 180,E1 -6770.262,E2 -6770.262} C_VEL
LIN {X 0,Y 482.415,Z 478.481,A -85,B 0,C 180,E1 -6771.359,E2 -6771.359} C_VEL
LIN {X 0,Y 482.845,Z 467.986,A -85,B 0,C 180,E1 -6772.35,E2 -6772.35} C_VEL
LIN {X 0,Y 483.384,Z 456.734,A -85,B 0,C 180,E1 -6773.192,E2 -6773.192} C_VEL
LIN {X 0,Y 483.749,Z 444.703,A -85,B 0,C 180,E1 -6773.9,E2 -6773.9} C_VEL
LIN {X 0,Y 484.03,Z 432.076,A -85,B 0,C 180,E1 -6774.445,E2 -6774.445} C_VEL
LIN {X 0,Y 484.16,Z 419.812,A -85,B 0,C 180,E1 -6774.809,E2 -6774.809} C_VEL
LIN {X 0,Y 484.476,Z 396.322,A -85,B 0,C 180,E1 -6775.193,E2 -6775.193} C_VEL
LIN {X 0,Y 485.036,Z 323.937,A -85,B 0,C 180,E1 -6776.275,E2 -6776.275} C_VEL
LIN {X 0,Y 482.349,Z 310.262,A -85,B 0,C 180,E1 -6776.61,E2 -6776.61} C_VEL
LIN {X 0,Y 482.582,Z 296.074,A -85,B 0,C 180,E1 -6779.335,E2 -6779.335} C_VEL
LIN {X 0,Y 481.703,Z 290.486,A -85,B 0,C 180,E1 -6780.511,E2 -6780.511} C_VEL
LIN {X 0,Y 481.697,Z 290.483,A -85,B 0,C 180,E1 -6783.733,E2 -6783.733} C_VEL
LIN {X 0,Y 481.625,Z 290.488,A -85,B 0,C 180,E1 -6786.747,E2 -6786.747} C_VEL
LIN {X 0,Y 481.676,Z 290.484,A -85,B 0,C 180,E1 -6789.94,E2 -6789.94} C_VEL
LIN {X 0,Y 481.637,Z 290.487,A -85,B 0,C 180,E1 -6793.3,E2 -6793.3} C_VEL
LIN {X 0,Y 481.653,Z 290.484,A -85,B 0,C 180,E1 -6795.641,E2 -6795.641} C_VEL
LIN {X 0,Y 481.655,Z 290.489,A -85,B 0,C 180,E1 -6798.958,E2 -6798.958} C_VEL
LIN {X 0,Y 481.653,Z 290.482,A -85,B 0,C 180,E1 -6801.993,E2 -6801.993} C_VEL
LIN {X 0,Y 481.688,Z 290.481,A -85,B 0,C 180,E1 -6805.318,E2 -6805.318} C_VEL
LIN {X 0,Y 481.643,Z 290.482,A -85,B 0,C 180,E1 -6808.312,E2 -6808.312} C_VEL
LIN {X 0,Y 481.699,Z 290.482,A -85,B 0,C 180,E1 -6811.219,E2 -6811.219} C_VEL
LIN {X 0,Y 481.696,Z 290.476,A -85,B 0,C 180,E1 -6814.043,E2 -6814.043} C_VEL
LIN {X 0,Y 481.673,Z 290.478,A -85,B 0,C 180,E1 -6816.812,E2 -6816.812} C_VEL
LIN {X 0,Y 481.694,Z 290.482,A -85,B 0,C 180,E1 -6819.503,E2 -6819.503} C_VEL
LIN {X 0,Y 481.703,Z 290.478,A -85,B 0,C 180,E1 -6822.158,E2 -6822.158} C_VEL
LIN {X 0,Y 481.742,Z 290.469,A -85,B 0,C 180,E1 -6824.776,E2 -6824.776} C_VEL
LIN {X 0,Y 481.75,Z 290.471,A -85,B 0,C 180,E1 -6828.215,E2 -6828.215} C_VEL
LIN {X 0,Y 481.762,Z 290.476,A -85,B 0,C 180,E1 -6831.612,E2 -6831.612} C_VEL
LIN {X 0,Y 481.806,Z 290.468,A -85,B 0,C 180,E1 -6834.14,E2 -6834.14} C_VEL
LIN {X 0,Y 481.927,Z 290.45,A -85,B 0,C 180,E1 -6837.493,E2 -6837.493} C_VEL
LIN {X 0,Y 481.885,Z 290.454,A -85,B 0,C 180,E1 -6840.836,E2 -6840.836} C_VEL
LIN {X 0,Y 481.927,Z 290.449,A -85,B 0,C 180,E1 -6842.508,E2 -6842.508} C_VEL
LIN {X 0,Y 481.807,Z 290.467,A -85,B 0,C 180,E1 -6845.861,E2 -6845.861} C_VEL
LIN {X 0,Y 481.762,Z 290.476,A -85,B 0,C 180,E1 -6848.388,E2 -6848.388} C_VEL
LIN {X 0,Y 481.75,Z 290.468,A -85,B 0,C 180,E1 -6851.785,E2 -6851.785} C_VEL
LIN {X 0,Y 481.742,Z 290.47,A -85,B 0,C 180,E1 -6855.224,E2 -6855.224} C_VEL
LIN {X 0,Y 481.712,Z 290.482,A -85,B 0,C 180,E1 -6858.722,E2 -6858.722} C_VEL
LIN {X 0,Y 481.645,Z 290.484,A -85,B 0,C 180,E1 -6861.395,E2 -6861.395} C_VEL
LIN {X 0,Y 481.674,Z 290.48,A -85,B 0,C 180,E1 -6864.113,E2 -6864.113} C_VEL
LIN {X 0,Y 481.747,Z 290.476,A -85,B 0,C 180,E1 -6867.139,E2 -6867.139} C_VEL
LIN {X 0,Y 481.679,Z 290.48,A -85,B 0,C 180,E1 -6869.741,E2 -6869.741} C_VEL
LIN {X 0,Y 481.672,Z 290.483,A -85,B 0,C 180,E1 -6872.674,E2 -6872.674} C_VEL
LIN {X 0,Y 481.637,Z 290.484,A -85,B 0,C 180,E1 -6875.71,E2 -6875.71} C_VEL
LIN {X 0,Y 481.672,Z 290.484,A -85,B 0,C 180,E1 -6878.859,E2 -6878.859} C_VEL
LIN {X 0,Y 481.654,Z 290.484,A -85,B 0,C 180,E1 -6881.913,E2 -6881.913} C_VEL
LIN {X 0,Y 481.656,Z 290.482,A -85,B 0,C 180,E1 -6884.458,E2 -6884.458} C_VEL
LIN {X 0,Y 481.649,Z 290.489,A -85,B 0,C 180,E1 -6887.839,E2 -6887.839} C_VEL
LIN {X 0,Y 481.663,Z 290.482,A -85,B 0,C 180,E1 -6890.654,E2 -6890.654} C_VEL
LIN {X 0,Y 481.629,Z 290.489,A -85,B 0,C 180,E1 -6893.376,E2 -6893.376} C_VEL
LIN {X 0,Y 481.712,Z 290.48,A -85,B 0,C 180,E1 -6896.33,E2 -6896.33} C_VEL
LIN {X 0,Y 481.653,Z 290.489,A -85,B 0,C 180,E1 -6899.418,E2 -6899.418} C_VEL
LIN {X 0,Y 481.702,Z 290.482,A -85,B 0,C 180,E1 -6902.168,E2 -6902.168} C_VEL
LIN {X 0,Y 481.735,Z 290.523,A -85,B 0,C 180,E1 -6904.272,E2 -6904.272} C_VEL
LIN {X 0,Y 483.752,Z 301.164,A -85,B 0,C 180,E1 -6906.245,E2 -6906.245} C_VEL
LIN {X 0,Y 483.441,Z 311.607,A -85,B 0,C 180,E1 -6908.034,E2 -6908.034} C_VEL
LIN {X 0,Y 482.729,Z 331.119,A -85,B 0,C 180,E1 -6911.319,E2 -6911.319} C_VEL
LIN {X 0,Y 482.247,Z 343.93,A -85,B 0,C 180,E1 -6913.446,E2 -6913.446} C_VEL
LIN {X 0,Y 484.898,Z 361.43,A -85,B 0,C 180,E1 -6913.815,E2 -6913.815} C_VEL
LIN {X 0,Y 484.272,Z 452.946,A -85,B 0,C 180,E1 -6915.207,E2 -6915.207} C_VEL
LIN {X 0,Y 483.952,Z 465.254,A -85,B 0,C 180,E1 -6915.546,E2 -6915.546} C_VEL
LIN {X 0,Y 483.526,Z 478.081,A -85,B 0,C 180,E1 -6916.07,E2 -6916.07} C_VEL
LIN {X 0,Y 483.06,Z 490.285,A -85,B 0,C 180,E1 -6916.753,E2 -6916.753} C_VEL
LIN {X 0,Y 482.601,Z 501.853,A -85,B 0,C 180,E1 -6917.596,E2 -6917.596} C_VEL
LIN {X 0,Y 482.191,Z 512.283,A -85,B 0,C 180,E1 -6918.546,E2 -6918.546} C_VEL
LIN {X 0,Y 481.817,Z 520.817,A -85,B 0,C 180,E1 -6919.494,E2 -6919.494} C_VEL
LIN {X 0,Y 481.472,Z 528.702,A -85,B 0,C 180,E1 -6920.548,E2 -6920.548} C_VEL
LIN {X 0,Y 481.226,Z 536.411,A -85,B 0,C 180,E1 -6921.813,E2 -6921.813} C_VEL
LIN {X 0,Y 481.006,Z 543.522,A -85,B 0,C 180,E1 -6923.287,E2 -6923.287} C_VEL
LIN {X 0,Y 480.931,Z 548.257,A -85,B 0,C 180,E1 -6924.549,E2 -6924.549} C_VEL
LIN {X 0,Y 480.829,Z 551.876,A -85,B 0,C 180,E1 -6925.809,E2 -6925.809} C_VEL
LIN {X 0,Y 480.888,Z 553.748,A -85,B 0,C 180,E1 -6926.648,E2 -6926.648} C_VEL
LIN {X 0,Y 480.821,Z 556.149,A -85,B 0,C 180,E1 -6928.325,E2 -6928.325} C_VEL
LIN {X 0,Y 480.745,Z 556.978,A -85,B 0,C 180,E1 -6930,E2 -6930} C_VEL
LIN {X 0,Y 480.821,Z 556.159,A -85,B 0,C 180,E1 -6931.675,E2 -6931.675} C_VEL
LIN {X 0,Y 480.888,Z 553.766,A -85,B 0,C 180,E1 -6933.351,E2 -6933.351} C_VEL
LIN {X 0,Y 480.838,Z 550.821,A -85,B 0,C 180,E1 -6934.611,E2 -6934.611} C_VEL
LIN {X 0,Y 480.925,Z 546.838,A -85,B 0,C 180,E1 -6935.871,E2 -6935.871} C_VEL
LIN {X 0,Y 481.106,Z 540.707,A -85,B 0,C 180,E1 -6937.343,E2 -6937.343} C_VEL
LIN {X 0,Y 481.311,Z 534.005,A -85,B 0,C 180,E1 -6938.607,E2 -6938.607} C_VEL
LIN {X 0,Y 481.593,Z 525.688,A -85,B 0,C 180,E1 -6939.873,E2 -6939.873} C_VEL
LIN {X 0,Y 481.977,Z 517.158,A -85,B 0,C 180,E1 -6940.927,E2 -6940.927} C_VEL
LIN {X 0,Y 482.428,Z 506.617,A -85,B 0,C 180,E1 -6941.981,E2 -6941.981} C_VEL
LIN {X 0,Y 482.866,Z 495.244,A -85,B 0,C 180,E1 -6942.893,E2 -6942.893} C_VEL
LIN {X 0,Y 483.248,Z 484.712,A -85,B 0,C 180,E1 -6943.562,E2 -6943.562} C_VEL
LIN {X 0,Y 483.663,Z 472.881,A -85,B 0,C 180,E1 -6944.14,E2 -6944.14} C_VEL
LIN {X 0,Y 483.984,Z 459.218,A -85,B 0,C 180,E1 -6944.613,E2 -6944.613} C_VEL
LIN {X 0,Y 484.276,Z 447.017,A -85,B 0,C 180,E1 -6944.873,E2 -6944.873} C_VEL
LIN {X 0,Y 484.795,Z 361.058,A -85,B 0,C 180,E1 -6946.151,E2 -6946.151} C_VEL
LIN {X 0,Y 482.254,Z 343.991,A -85,B 0,C 180,E1 -6946.51,E2 -6946.51} C_VEL
LIN {X 0,Y 482.845,Z 325.581,A -85,B 0,C 180,E1 -6949.558,E2 -6949.558} C_VEL
LIN {X 0,Y 483.53,Z 307.083,A -85,B 0,C 180,E1 -6952.654,E2 -6952.654} C_VEL
LIN {X 0,Y 483.655,Z 300.742,A -85,B 0,C 180,E1 -6953.729,E2 -6953.729} C_VEL
LIN {X 0,Y 481.75,Z 290.479,A -85,B 0,C 180,E1 -6955.6,E2 -6955.6} C_VEL
LIN {X 0,Y 481.701,Z 290.485,A -85,B 0,C 180,E1 -6957.831,E2 -6957.831} C_VEL
LIN {X 0,Y 481.645,Z 290.486,A -85,B 0,C 180,E1 -6960.71,E2 -6960.71} C_VEL
LIN {X 0,Y 481.697,Z 290.48,A -85,B 0,C 180,E1 -6963.732,E2 -6963.732} C_VEL
LIN {X 0,Y 481.624,Z 290.489,A -85,B 0,C 180,E1 -6966.746,E2 -6966.746} C_VEL
LIN {X 0,Y 481.675,Z 290.483,A -85,B 0,C 180,E1 -6969.94,E2 -6969.94} C_VEL
LIN {X 0,Y 481.636,Z 290.485,A -85,B 0,C 180,E1 -6973.299,E2 -6973.299} C_VEL
LIN {X 0,Y 481.651,Z 290.483,A -85,B 0,C 180,E1 -6975.641,E2 -6975.641} C_VEL
LIN {X 0,Y 481.654,Z 290.486,A -85,B 0,C 180,E1 -6978.958,E2 -6978.958} C_VEL
LIN {X 0,Y 481.651,Z 290.484,A -85,B 0,C 180,E1 -6981.992,E2 -6981.992} C_VEL
LIN {X 0,Y 481.685,Z 290.481,A -85,B 0,C 180,E1 -6985.317,E2 -6985.317} C_VEL
LIN {X 0,Y 481.641,Z 290.486,A -85,B 0,C 180,E1 -6988.311,E2 -6988.311} C_VEL
LIN {X 0,Y 481.696,Z 290.482,A -85,B 0,C 180,E1 -6991.218,E2 -6991.218} C_VEL
LIN {X 0,Y 481.697,Z 290.477,A -85,B 0,C 180,E1 -6994.042,E2 -6994.042} C_VEL
LIN {X 0,Y 481.67,Z 290.485,A -85,B 0,C 180,E1 -6996.811,E2 -6996.811} C_VEL
LIN {X 0,Y 481.691,Z 290.482,A -85,B 0,C 180,E1 -6999.502,E2 -6999.502} C_VEL
LIN {X 0,Y 481.702,Z 290.476,A -85,B 0,C 180,E1 -7002.158,E2 -7002.158} C_VEL
LIN {X 0,Y 481.739,Z 290.474,A -85,B 0,C 180,E1 -7004.775,E2 -7004.775} C_VEL
LIN {X 0,Y 481.746,Z 290.471,A -85,B 0,C 180,E1 -7008.215,E2 -7008.215} C_VEL
LIN {X 0,Y 481.758,Z 290.477,A -85,B 0,C 180,E1 -7011.611,E2 -7011.611} C_VEL
LIN {X 0,Y 481.808,Z 290.465,A -85,B 0,C 180,E1 -7014.139,E2 -7014.139} C_VEL
LIN {X 0,Y 481.921,Z 290.456,A -85,B 0,C 180,E1 -7017.492,E2 -7017.492} C_VEL
LIN {X 0,Y 481.934,Z 290.453,A -85,B 0,C 180,E1 -7020,E2 -7020} C_VEL
LIN {X 0,Y 481.922,Z 290.45,A -85,B 0,C 180,E1 -7022.507,E2 -7022.507} C_VEL
LIN {X 0,Y 481.793,Z 290.474,A -85,B 0,C 180,E1 -7025.861,E2 -7025.861} C_VEL
LIN {X 0,Y 481.757,Z 290.473,A -85,B 0,C 180,E1 -7028.388,E2 -7028.388} C_VEL
LIN {X 0,Y 481.745,Z 290.476,A -85,B 0,C 180,E1 -7031.785,E2 -7031.785} C_VEL
LIN {X 0,Y 481.736,Z 290.472,A -85,B 0,C 180,E1 -7035.224,E2 -7035.224} C_VEL
LIN {X 0,Y 481.702,Z 290.479,A -85,B 0,C 180,E1 -7038.722,E2 -7038.722} C_VEL
LIN {X 0,Y 481.639,Z 290.484,A -85,B 0,C 180,E1 -7041.395,E2 -7041.395} C_VEL
LIN {X 0,Y 481.655,Z 290.487,A -85,B 0,C 180,E1 -7044.114,E2 -7044.114} C_VEL
LIN {X 0,Y 481.711,Z 290.476,A -85,B 0,C 180,E1 -7047.132,E2 -7047.132} C_VEL
LIN {X 0,Y 481.672,Z 290.481,A -85,B 0,C 180,E1 -7049.741,E2 -7049.741} C_VEL
LIN {X 0,Y 481.666,Z 290.489,A -85,B 0,C 180,E1 -7052.674,E2 -7052.674} C_VEL
LIN {X 0,Y 481.631,Z 290.485,A -85,B 0,C 180,E1 -7055.71,E2 -7055.71} C_VEL
LIN {X 0,Y 481.663,Z 290.49,A -85,B 0,C 180,E1 -7058.86,E2 -7058.86} C_VEL
LIN {X 0,Y 481.647,Z 290.483,A -85,B 0,C 180,E1 -7061.913,E2 -7061.913} C_VEL
LIN {X 0,Y 481.655,Z 290.485,A -85,B 0,C 180,E1 -7064.458,E2 -7064.458} C_VEL
LIN {X 0,Y 481.624,Z 290.486,A -85,B 0,C 180,E1 -7067.838,E2 -7067.838} C_VEL
LIN {X 0,Y 481.662,Z 290.491,A -85,B 0,C 180,E1 -7071.141,E2 -7071.141} C_VEL
LIN {X 0,Y 481.632,Z 290.485,A -85,B 0,C 180,E1 -7074.291,E2 -7074.291} C_VEL
LIN {X 0,Y 481.667,Z 290.49,A -85,B 0,C 180,E1 -7077.326,E2 -7077.326} C_VEL
LIN {X 0,Y 481.665,Z 290.481,A -85,B 0,C 180,E1 -7080.259,E2 -7080.259} C_VEL
LIN {X 0,Y 481.657,Z 290.486,A -85,B 0,C 180,E1 -7083.107,E2 -7083.107} C_VEL
LIN {X 0,Y 481.645,Z 290.487,A -85,B 0,C 180,E1 -7085.886,E2 -7085.886} C_VEL
LIN {X 0,Y 481.634,Z 290.489,A -85,B 0,C 180,E1 -7087.963,E2 -7087.963} C_VEL
LIN {X 0,Y 480.966,Z 290.569,A -85,B 0,C 180,E1 -7088.661,E2 -7088.661} C_VEL
LIN {X 0,Y 478.142,Z 290.927,A -85,B 0,C 180,E1 -7089.796,E2 -7089.796} C_VEL
LIN {X 0,Y 475.756,Z 291.223,A -85,B 0,C 180,E1 -7090.71,E2 -7090.71} C_VEL
LIN {X 0,Y 474.727,Z 291.351,A -85,B 0,C 180,E1 -7091.416,E2 -7091.416} C_VEL
LIN {X 0,Y 474.641,Z 291.361,A -85,B 0,C 180,E1 -7091.655,E2 -7091.655} C_VEL
LIN {X 0,Y 474.698,Z 291.349,A -85,B 0,C 180,E1 -7094.545,E2 -7094.545} C_VEL
LIN {X 0,Y 474.691,Z 291.359,A -85,B 0,C 180,E1 -7098.038,E2 -7098.038} C_VEL
LIN {X 0,Y 474.656,Z 291.496,A -85,B 0,C 180,E1 -7099.523,E2 -7099.523} C_VEL
LIN {X 0,Y 475.564,Z 297.989,A -85,B 0,C 180,E1 -7100.859,E2 -7100.859} C_VEL
LIN {X 0,Y 475.346,Z 310.617,A -85,B 0,C 180,E1 -7103.341,E2 -7103.341} C_VEL
LIN {X 0,Y 478.134,Z 325.587,A -85,B 0,C 180,E1 -7103.671,E2 -7103.671} C_VEL
LIN {X 0,Y 477.347,Z 418.469,A -85,B 0,C 180,E1 -7105.091,E2 -7105.091} C_VEL
LIN {X 0,Y 477.069,Z 432.097,A -85,B 0,C 180,E1 -7105.485,E2 -7105.485} C_VEL
LIN {X 0,Y 476.8,Z 444.832,A -85,B 0,C 180,E1 -7106.038,E2 -7106.038} C_VEL
LIN {X 0,Y 476.397,Z 456.477,A -85,B 0,C 180,E1 -7106.723,E2 -7106.723} C_VEL
LIN {X 0,Y 475.832,Z 467.731,A -85,B 0,C 180,E1 -7107.567,E2 -7107.567} C_VEL
LIN {X 0,Y 475.339,Z 477.881,A -85,B 0,C 180,E1 -7108.518,E2 -7108.518} C_VEL
LIN {X 0,Y 475.004,Z 486.992,A -85,B 0,C 180,E1 -7109.576,E2 -7109.576} C_VEL
LIN {X 0,Y 474.609,Z 495.871,A -85,B 0,C 180,E1 -7110.849,E2 -7110.849} C_VEL
LIN {X 0,Y 474.27,Z 503.047,A -85,B 0,C 180,E1 -7112.123,E2 -7112.123} C_VEL
LIN {X 0,Y 474.093,Z 508.789,A -85,B 0,C 180,E1 -7113.4,E2 -7113.4} C_VEL
LIN {X 0,Y 473.874,Z 513.33,A -85,B 0,C 180,E1 -7114.679,E2 -7114.679} C_VEL
LIN {X 0,Y 473.894,Z 516.778,A -85,B 0,C 180,E1 -7115.959,E2 -7115.959} C_VEL
LIN {X 0,Y 473.829,Z 518.516,A -85,B 0,C 180,E1 -7116.815,E2 -7116.815} C_VEL
LIN {X 0,Y 473.717,Z 520.771,A -85,B 0,C 180,E1 -7118.532,E2 -7118.532} C_VEL
LIN {X 0,Y 473.653,Z 521.304,A -85,B 0,C 180,E1 -7119.394,E2 -7119.394} C_VEL
LIN {X 0,Y 473.69,Z 521.396,A -85,B 0,C 180,E1 -7120.256,E2 -7120.256} C_VEL
LIN {X 0,Y 473.759,Z 520.635,A -85,B 0,C 180,E1 -7121.741,E2 -7121.741} C_VEL
LIN {X 0,Y 473.704,Z 519.294,A -85,B 0,C 180,E1 -7122.859,E2 -7122.859} C_VEL
LIN {X 0,Y 473.82,Z 516.799,A -85,B 0,C 180,E1 -7124.167,E2 -7124.167} C_VEL
LIN {X 0,Y 473.972,Z 513.25,A -85,B 0,C 180,E1 -7125.48,E2 -7125.48} C_VEL
LIN {X 0,Y 474.104,Z 508.527,A -85,B 0,C 180,E1 -7126.802,E2 -7126.802} C_VEL
LIN {X 0,Y 474.385,Z 502.477,A -85,B 0,C 180,E1 -7128.127,E2 -7128.127} C_VEL
LIN {X 0,Y 474.725,Z 494.863,A -85,B 0,C 180,E1 -7129.457,E2 -7129.457} C_VEL
LIN {X 0,Y 475.056,Z 487.022,A -85,B 0,C 180,E1 -7130.571,E2 -7130.571} C_VEL
LIN {X 0,Y 475.553,Z 477.393,A -85,B 0,C 180,E1 -7131.683,E2 -7131.683} C_VEL
LIN {X 0,Y 476.048,Z 466.561,A -85,B 0,C 180,E1 -7132.687,E2 -7132.687} C_VEL
LIN {X 0,Y 476.541,Z 456.063,A -85,B 0,C 180,E1 -7133.465,E2 -7133.465} C_VEL
LIN {X 0,Y 476.889,Z 444.193,A -85,B 0,C 180,E1 -7134.16,E2 -7134.16} C_VEL
LIN {X 0,Y 477.238,Z 431.542,A -85,B 0,C 180,E1 -7134.7,E2 -7134.7} C_VEL
LIN {X 0,Y 477.42,Z 418.926,A -85,B 0,C 180,E1 -7135.067,E2 -7135.067} C_VEL
LIN {X 0,Y 477.98,Z 361.433,A -85,B 0,C 180,E1 -7135.964,E2 -7135.964} C_VEL
LIN {X 0,Y 478.232,Z 324.683,A -85,B 0,C 180,E1 -7136.525,E2 -7136.525} C_VEL
LIN {X 0,Y 475.4,Z 310.575,A -85,B 0,C 180,E1 -7136.869,E2 -7136.869} C_VEL
LIN {X 0,Y 475.671,Z 297.813,A -85,B 0,C 180,E1 -7139.341,E2 -7139.341} C_VEL
LIN {X 0,Y 474.635,Z 291.365,A -85,B 0,C 180,E1 -7140.68,E2 -7140.68} C_VEL
LIN {X 0,Y 474.637,Z 291.365,A -85,B 0,C 180,E1 -7143.984,E2 -7143.984} C_VEL
LIN {X 0,Y 474.571,Z 291.365,A -85,B 0,C 180,E1 -7146.899,E2 -7146.899} C_VEL
LIN {X 0,Y 474.617,Z 291.362,A -85,B 0,C 180,E1 -7149.646,E2 -7149.646} C_VEL
LIN {X 0,Y 474.613,Z 291.365,A -85,B 0,C 180,E1 -7152.934,E2 -7152.934} C_VEL
LIN {X 0,Y 474.605,Z 291.363,A -85,B 0,C 180,E1 -7155.895,E2 -7155.895} C_VEL
LIN {X 0,Y 474.627,Z 291.363,A -85,B 0,C 180,E1 -7159.041,E2 -7159.041} C_VEL
LIN {X 0,Y 474.609,Z 291.359,A -85,B 0,C 180,E1 -7161.704,E2 -7161.704} C_VEL
LIN {X 0,Y 474.624,Z 291.363,A -85,B 0,C 180,E1 -7164.726,E2 -7164.726} C_VEL
LIN {X 0,Y 474.634,Z 291.355,A -85,B 0,C 180,E1 -7167.788,E2 -7167.788} C_VEL
LIN {X 0,Y 474.623,Z 291.361,A -85,B 0,C 180,E1 -7170.885,E2 -7170.885} C_VEL
LIN {X 0,Y 474.657,Z 291.356,A -85,B 0,C 180,E1 -7173.628,E2 -7173.628} C_VEL
LIN {X 0,Y 474.635,Z 291.354,A -85,B 0,C 180,E1 -7176.641,E2 -7176.641} C_VEL
LIN {X 0,Y 474.653,Z 291.352,A -85,B 0,C 180,E1 -7180.09,E2 -7180.09} C_VEL
LIN {X 0,Y 474.647,Z 291.357,A -85,B 0,C 180,E1 -7182.775,E2 -7182.775} C_VEL
LIN {X 0,Y 474.647,Z 291.359,A -85,B 0,C 180,E1 -7185.421,E2 -7185.421} C_VEL
LIN {X 0,Y 474.703,Z 291.35,A -85,B 0,C 180,E1 -7188.038,E2 -7188.038} C_VEL
LIN {X 0,Y 474.727,Z 291.351,A -85,B 0,C 180,E1 -7191.487,E2 -7191.487} C_VEL
LIN {X 0,Y 474.769,Z 291.346,A -85,B 0,C 180,E1 -7194.052,E2 -7194.052} C_VEL
LIN {X 0,Y 474.893,Z 291.326,A -85,B 0,C 180,E1 -7197.456,E2 -7197.456} C_VEL
LIN {X 0,Y 474.911,Z 291.33,A -85,B 0,C 180,E1 -7200,E2 -7200} C_VEL
LIN {X 0,Y 474.893,Z 291.325,A -85,B 0,C 180,E1 -7202.545,E2 -7202.545} C_VEL
LIN {X 0,Y 474.769,Z 291.345,A -85,B 0,C 180,E1 -7205.948,E2 -7205.948} C_VEL
LIN {X 0,Y 474.727,Z 291.351,A -85,B 0,C 180,E1 -7208.514,E2 -7208.514} C_VEL
LIN {X 0,Y 474.704,Z 291.348,A -85,B 0,C 180,E1 -7211.963,E2 -7211.963} C_VEL
LIN {X 0,Y 474.7,Z 291.346,A -85,B 0,C 180,E1 -7215.456,E2 -7215.456} C_VEL
LIN {X 0,Y 474.665,Z 291.355,A -85,B 0,C 180,E1 -7219.01,E2 -7219.01} C_VEL
LIN {X 0,Y 474.588,Z 291.362,A -85,B 0,C 180,E1 -7221.729,E2 -7221.729} C_VEL
LIN {X 0,Y 474.657,Z 291.358,A -85,B 0,C 180,E1 -7224.493,E2 -7224.493} C_VEL
LIN {X 0,Y 474.681,Z 291.353,A -85,B 0,C 180,E1 -7227.335,E2 -7227.335} C_VEL
LIN {X 0,Y 474.605,Z 291.362,A -85,B 0,C 180,E1 -7230.23,E2 -7230.23} C_VEL
LIN {X 0,Y 474.643,Z 291.363,A -85,B 0,C 180,E1 -7233.22,E2 -7233.22} C_VEL
LIN {X 0,Y 474.589,Z 291.361,A -85,B 0,C 180,E1 -7236.324,E2 -7236.324} C_VEL
LIN {X 0,Y 474.619,Z 291.354,A -85,B 0,C 180,E1 -7239.646,E2 -7239.646} C_VEL
LIN {X 0,Y 474.616,Z 291.362,A -85,B 0,C 180,E1 -7242.934,E2 -7242.934} C_VEL
LIN {X 0,Y 474.606,Z 291.364,A -85,B 0,C 180,E1 -7245.895,E2 -7245.895} C_VEL
LIN {X 0,Y 474.629,Z 291.361,A -85,B 0,C 180,E1 -7249.041,E2 -7249.041} C_VEL
LIN {X 0,Y 474.611,Z 291.367,A -85,B 0,C 180,E1 -7251.704,E2 -7251.704} C_VEL
LIN {X 0,Y 474.626,Z 291.36,A -85,B 0,C 180,E1 -7254.726,E2 -7254.726} C_VEL
LIN {X 0,Y 474.638,Z 291.363,A -85,B 0,C 180,E1 -7257.788,E2 -7257.788} C_VEL
LIN {X 0,Y 474.626,Z 291.362,A -85,B 0,C 180,E1 -7260.885,E2 -7260.885} C_VEL
LIN {X 0,Y 474.674,Z 291.356,A -85,B 0,C 180,E1 -7263.629,E2 -7263.629} C_VEL
LIN {X 0,Y 474.703,Z 291.438,A -85,B 0,C 180,E1 -7264.045,E2 -7264.045} C_VEL
LIN {X 0,Y 476.874,Z 302.857,A -85,B 0,C 180,E1 -7266.2,E2 -7266.2} C_VEL
LIN {X 0,Y 476.365,Z 316.013,A -85,B 0,C 180,E1 -7268.48,E2 -7268.48} C_VEL
LIN {X 0,Y 475.635,Z 334.889,A -85,B 0,C 180,E1 -7271.7,E2 -7271.7} C_VEL
LIN {X 0,Y 475.297,Z 343.683,A -85,B 0,C 180,E1 -7273.182,E2 -7273.182} C_VEL
LIN {X 0,Y 478.117,Z 362.247,A -85,B 0,C 180,E1 -7273.579,E2 -7273.579} C_VEL
LIN {X 0,Y 477.452,Z 452.193,A -85,B 0,C 180,E1 -7274.963,E2 -7274.963} C_VEL
LIN {X 0,Y 477.118,Z 463.89,A -85,B 0,C 180,E1 -7275.28,E2 -7275.28} C_VEL
LIN {X 0,Y 476.678,Z 476.984,A -85,B 0,C 180,E1 -7275.811,E2 -7275.811} C_VEL
LIN {X 0,Y 476.214,Z 488.568,A -85,B 0,C 180,E1 -7276.45,E2 -7276.45} C_VEL
LIN {X 0,Y 475.785,Z 499.147,A -85,B 0,C 180,E1 -7277.199,E2 -7277.199} C_VEL
LIN {X 0,Y 475.327,Z 509.993,A -85,B 0,C 180,E1 -7278.161,E2 -7278.161} C_VEL
LIN {X 0,Y 474.814,Z 520.644,A -85,B 0,C 180,E1 -7279.338,E2 -7279.338} C_VEL
LIN {X 0,Y 474.37,Z 529.878,A -85,B 0,C 180,E1 -7280.62,E2 -7280.62} C_VEL
LIN {X 0,Y 474.114,Z 537.314,A -85,B 0,C 180,E1 -7281.904,E2 -7281.904} C_VEL
LIN {X 0,Y 473.922,Z 543.29,A -85,B 0,C 180,E1 -7283.186,E2 -7283.186} C_VEL
LIN {X 0,Y 473.845,Z 548.016,A -85,B 0,C 180,E1 -7284.467,E2 -7284.467} C_VEL
LIN {X 0,Y 473.735,Z 551.627,A -85,B 0,C 180,E1 -7285.746,E2 -7285.746} C_VEL
LIN {X 0,Y 473.795,Z 553.493,A -85,B 0,C 180,E1 -7286.598,E2 -7286.598} C_VEL
LIN {X 0,Y 473.724,Z 555.89,A -85,B 0,C 180,E1 -7288.299,E2 -7288.299} C_VEL
LIN {X 0,Y 473.689,Z 556.499,A -85,B 0,C 180,E1 -7289.15,E2 -7289.15} C_VEL
LIN {X 0,Y 473.672,Z 556.714,A -85,B 0,C 180,E1 -7290,E2 -7290} C_VEL
LIN {X 0,Y 473.724,Z 555.89,A -85,B 0,C 180,E1 -7291.7,E2 -7291.7} C_VEL
LIN {X 0,Y 473.741,Z 554.892,A -85,B 0,C 180,E1 -7292.55,E2 -7292.55} C_VEL
LIN {X 0,Y 473.795,Z 553.491,A -85,B 0,C 180,E1 -7293.401,E2 -7293.401} C_VEL
LIN {X 0,Y 473.762,Z 550.541,A -85,B 0,C 180,E1 -7294.68,E2 -7294.68} C_VEL
LIN {X 0,Y 473.832,Z 546.547,A -85,B 0,C 180,E1 -7295.959,E2 -7295.959} C_VEL
LIN {X 0,Y 474.015,Z 540.401,A -85,B 0,C 180,E1 -7297.454,E2 -7297.454} C_VEL
LIN {X 0,Y 474.242,Z 533.686,A -85,B 0,C 180,E1 -7298.737,E2 -7298.737} C_VEL
LIN {X 0,Y 474.556,Z 525.352,A -85,B 0,C 180,E1 -7300.021,E2 -7300.021} C_VEL
LIN {X 0,Y 474.978,Z 516.796,A -85,B 0,C 180,E1 -7301.09,E2 -7301.09} C_VEL
LIN {X 0,Y 475.441,Z 506.424,A -85,B 0,C 180,E1 -7302.141,E2 -7302.141} C_VEL
LIN {X 0,Y 475.857,Z 496.03,A -85,B 0,C 180,E1 -7302.994,E2 -7302.994} C_VEL
LIN {X 0,Y 476.321,Z 484.219,A -85,B 0,C 180,E1 -7303.763,E2 -7303.763} C_VEL
LIN {X 0,Y 476.758,Z 472.283,A -85,B 0,C 180,E1 -7304.349,E2 -7304.349} C_VEL
LIN {X 0,Y 477.124,Z 458.475,A -85,B 0,C 180,E1 -7304.828,E2 -7304.828} C_VEL
LIN {X 0,Y 477.385,Z 445.868,A -85,B 0,C 180,E1 -7305.093,E2 -7305.093} C_VEL
LIN {X 0,Y 477.934,Z 361.708,A -85,B 0,C 180,E1 -7306.36,E2 -7306.36} C_VEL
LIN {X 0,Y 475.238,Z 343.859,A -85,B 0,C 180,E1 -7306.721,E2 -7306.721} C_VEL
LIN {X 0,Y 475.909,Z 325.192,A -85,B 0,C 180,E1 -7309.855,E2 -7309.855} C_VEL
LIN {X 0,Y 476.652,Z 306.676,A -85,B 0,C 180,E1 -7312.999,E2 -7312.999} C_VEL
LIN {X 0,Y 476.611,Z 301.472,A -85,B 0,C 180,E1 -7313.902,E2 -7313.902} C_VEL
LIN {X 0,Y 474.705,Z 291.357,A -85,B 0,C 180,E1 -7315.766,E2 -7315.766} C_VEL
LIN {X 0,Y 474.646,Z 291.365,A -85,B 0,C 180,E1 -7318.282,E2 -7318.282} C_VEL
LIN {X 0,Y 474.598,Z 291.362,A -85,B 0,C 180,E1 -7321.217,E2 -7321.217} C_VEL
LIN {X 0,Y 474.632,Z 291.366,A -85,B 0,C 180,E1 -7324.24,E2 -7324.24} C_VEL
LIN {X 0,Y 474.589,Z 291.363,A -85,B 0,C 180,E1 -7327.383,E2 -7327.383} C_VEL
LIN {X 0,Y 474.616,Z 291.364,A -85,B 0,C 180,E1 -7330.657,E2 -7330.657} C_VEL
LIN {X 0,Y 474.598,Z 291.361,A -85,B 0,C 180,E1 -7333.48,E2 -7333.48} C_VEL
LIN {X 0,Y 474.598,Z 291.371,A -85,B 0,C 180,E1 -7336.518,E2 -7336.518} C_VEL
LIN {X 0,Y 474.615,Z 291.36,A -85,B 0,C 180,E1 -7339.342,E2 -7339.342} C_VEL
LIN {X 0,Y 474.607,Z 291.36,A -85,B 0,C 180,E1 -7341.703,E2 -7341.703} C_VEL
LIN {X 0,Y 474.622,Z 291.367,A -85,B 0,C 180,E1 -7344.725,E2 -7344.725} C_VEL
LIN {X 0,Y 474.632,Z 291.357,A -85,B 0,C 180,E1 -7347.787,E2 -7347.787} C_VEL
LIN {X 0,Y 474.621,Z 291.367,A -85,B 0,C 180,E1 -7350.884,E2 -7350.884} C_VEL
LIN {X 0,Y 474.656,Z 291.356,A -85,B 0,C 180,E1 -7353.628,E2 -7353.628} C_VEL
LIN {X 0,Y 474.632,Z 291.36,A -85,B 0,C 180,E1 -7356.641,E2 -7356.641} C_VEL
LIN {X 0,Y 474.65,Z 291.355,A -85,B 0,C 180,E1 -7360.089,E2 -7360.089} C_VEL
LIN {X 0,Y 474.646,Z 291.358,A -85,B 0,C 180,E1 -7362.774,E2 -7362.774} C_VEL
LIN {X 0,Y 474.647,Z 291.363,A -85,B 0,C 180,E1 -7365.421,E2 -7365.421} C_VEL
LIN {X 0,Y 474.699,Z 291.35,A -85,B 0,C 180,E1 -7368.037,E2 -7368.037} C_VEL
